# B&R Automation Studio project TD52 (part 17)

```c
/* Source: slatzm.f */
#define slatzm FORTRAN_WRAPPER(slatzm)
extern void slatzm(
    char   *side,
    ptrdiff_t *m,
    ptrdiff_t *n,
    float  *v,
    ptrdiff_t *incv,
    float  *tau,
    float  *c1,
    float  *c2,
    ptrdiff_t *ldc,
    float  *work
);

/* Source: slauu2.f */
#define slauu2 FORTRAN_WRAPPER(slauu2)
extern void slauu2(
    char   *uplo,
    ptrdiff_t *n,
    float  *a,
    ptrdiff_t *lda,
    ptrdiff_t *info
);

/* Source: slauum.f */
#define slauum FORTRAN_WRAPPER(slauum)
extern void slauum(
    char   *uplo,
    ptrdiff_t *n,
    float  *a,
    ptrdiff_t *lda,
    ptrdiff_t *info
);

/* Source: sopgtr.f */
#define sopgtr FORTRAN_WRAPPER(sopgtr)
extern void sopgtr(
    char   *uplo,
    ptrdiff_t *n,
    float  *ap,
    float  *tau,
    float  *q,
    ptrdiff_t *ldq,
    float  *work,
    ptrdiff_t *info
);

/* Source: sopmtr.f */
#define sopmtr FORTRAN_WRAPPER(sopmtr)
extern void sopmtr(
    char   *side,
    char   *uplo,
    char   *trans,
    ptrdiff_t *m,
    ptrdiff_t *n,
    float  *ap,
    float  *tau,
    float  *c,
    ptrdiff_t *ldc,
    float  *work,
    ptrdiff_t *info
);

/* Source: sorg2l.f */
#define sorg2l FORTRAN_WRAPPER(sorg2l)
extern void sorg2l(
    ptrdiff_t *m,
    ptrdiff_t *n,
    ptrdiff_t *k,
    float  *a,
    ptrdiff_t *lda,
    float  *tau,
    float  *work,
    ptrdiff_t *info
);

/* Source: sorg2r.f */
#define sorg2r FORTRAN_WRAPPER(sorg2r)
extern void sorg2r(
    ptrdiff_t *m,
    ptrdiff_t *n,
    ptrdiff_t *k,
    float  *a,
    ptrdiff_t *lda,
    float  *tau,
    float  *work,
    ptrdiff_t *info
);

/* Source: sorgbr.f */
#define sorgbr FORTRAN_WRAPPER(sorgbr)
extern void sorgbr(
    char   *vect,
    ptrdiff_t *m,
    ptrdiff_t *n,
    ptrdiff_t *k,
    float  *a,
    ptrdiff_t *lda,
    float  *tau,
    float  *work,
    ptrdiff_t *lwork,
    ptrdiff_t *info
);

/* Source: sorghr.f */
#define sorghr FORTRAN_WRAPPER(sorghr)
extern void sorghr(
    ptrdiff_t *n,
    ptrdiff_t *ilo,
    ptrdiff_t *ihi,
    float  *a,
    ptrdiff_t *lda,
    float  *tau,
    float  *work,
    ptrdiff_t *lwork,
    ptrdiff_t *info
);

/* Source: sorgl2.f */
#define sorgl2 FORTRAN_WRAPPER(sorgl2)
extern void sorgl2(
    ptrdiff_t *m,
    ptrdiff_t *n,
    ptrdiff_t *k,
    float  *a,
    ptrdiff_t *lda,
    float  *tau,
    float  *work,
    ptrdiff_t *info
);

/* Source: sorglq.f */
#define sorglq FORTRAN_WRAPPER(sorglq)
extern void sorglq(
    ptrdiff_t *m,
    ptrdiff_t *n,
    ptrdiff_t *k,
    float  *a,
    ptrdiff_t *lda,
    float  *tau,
    float  *work,
    ptrdiff_t *lwork,
    ptrdiff_t *info
);

/* Source: sorgql.f */
#define sorgql FORTRAN_WRAPPER(sorgql)
extern void sorgql(
    ptrdiff_t *m,
    ptrdiff_t *n,
    ptrdiff_t *k,
    float  *a,
    ptrdiff_t *lda,
    float  *tau,
    float  *work,
    ptrdiff_t *lwork,
    ptrdiff_t *info
);

/* Source: sorgqr.f */
#define sorgqr FORTRAN_WRAPPER(sorgqr)
extern void sorgqr(
    ptrdiff_t *m,
    ptrdiff_t *n,
    ptrdiff_t *k,
    float  *a,
    ptrdiff_t *lda,
    float  *tau,
    float  *work,
    ptrdiff_t *lwork,
    ptrdiff_t *info
);

/* Source: sorgr2.f */
#define sorgr2 FORTRAN_WRAPPER(sorgr2)
extern void sorgr2(
    ptrdiff_t *m,
    ptrdiff_t *n,
    ptrdiff_t *k,
    float  *a,
    ptrdiff_t *lda,
    float  *tau,
    float  *work,
    ptrdiff_t *info
);

/* Source: sorgrq.f */
#define sorgrq FORTRAN_WRAPPER(sorgrq)
extern void sorgrq(
    ptrdiff_t *m,
    ptrdiff_t *n,
    ptrdiff_t *k,
    float  *a,
    ptrdiff_t *lda,
    float  *tau,
    float  *work,
    ptrdiff_t *lwork,
    ptrdiff_t *info
);

/* Source: sorgtr.f */
#define sorgtr FORTRAN_WRAPPER(sorgtr)
extern void sorgtr(
    char   *uplo,
    ptrdiff_t *n,
    float  *a,
    ptrdiff_t *lda,
    float  *tau,
    float  *work,
    ptrdiff_t *lwork,
    ptrdiff_t *info
);

/* Source: sorm2l.f */
#define sorm2l FORTRAN_WRAPPER(sorm2l)
extern void sorm2l(
    char   *side,
    char   *trans,
    ptrdiff_t *m,
    ptrdiff_t *n,
    ptrdiff_t *k,
    float  *a,
    ptrdiff_t *lda,
    float  *tau,
    float  *c,
    ptrdiff_t *ldc,
    float  *work,
    ptrdiff_t *info
);

/* Source: sorm2r.f */
#define sorm2r FORTRAN_WRAPPER(sorm2r)
extern void sorm2r(
    char   *side,
    char   *trans,
    ptrdiff_t *m,
    ptrdiff_t *n,
    ptrdiff_t *k,
    float  *a,
    ptrdiff_t *lda,
    float  *tau,
    float  *c,
    ptrdiff_t *ldc,
    float  *work,
    ptrdiff_t *info
);

/* Source: sormbr.f */
#define sormbr FORTRAN_WRAPPER(sormbr)
extern void sormbr(
    char   *vect,
    char   *side,
    char   *trans,
    ptrdiff_t *m,
    ptrdiff_t *n,
    ptrdiff_t *k,
    float  *a,
    ptrdiff_t *lda,
    float  *tau,
    float  *c,
    ptrdiff_t *ldc,
    float  *work,
    ptrdiff_t *lwork,
    ptrdiff_t *info
);

/* Source: sormhr.f */
#define sormhr FORTRAN_WRAPPER(sormhr)
extern void sormhr(
    char   *side,
    char   *trans,
    ptrdiff_t *m,
    ptrdiff_t *n,
    ptrdiff_t *ilo,
    ptrdiff_t *ihi,
    float  *a,
    ptrdiff_t *lda,
    float  *tau,
    float  *c,
    ptrdiff_t *ldc,
    float  *work,
    ptrdiff_t *lwork,
    ptrdiff_t *info
);

/* Source: sorml2.f */
#define sorml2 FORTRAN_WRAPPER(sorml2)
extern void sorml2(
    char   *side,
    char   *trans,
    ptrdiff_t *m,
    ptrdiff_t *n,
    ptrdiff_t *k,
    float  *a,
    ptrdiff_t *lda,
    float  *tau,
    float  *c,
    ptrdiff_t *ldc,
    float  *work,
    ptrdiff_t *info
);

/* Source: sormlq.f */
#define sormlq FORTRAN_WRAPPER(sormlq)
extern void sormlq(
    char   *side,
    char   *trans,
    ptrdiff_t *m,
    ptrdiff_t *n,
    ptrdiff_t *k,
    float  *a,
    ptrdiff_t *lda,
    float  *tau,
    float  *c,
    ptrdiff_t *ldc,
    float  *work,
    ptrdiff_t *lwork,
    ptrdiff_t *info
);

/* Source: sormql.f */
#define sormql FORTRAN_WRAPPER(sormql)
extern void sormql(
    char   *side,
    char   *trans,
    ptrdiff_t *m,
    ptrdiff_t *n,
    ptrdiff_t *k,
    float  *a,
    ptrdiff_t *lda,
    float  *tau,
    float  *c,
    ptrdiff_t *ldc,
    float  *work,
    ptrdiff_t *lwork,
    ptrdiff_t *info
);

/* Source: sormqr.f */
#define sormqr FORTRAN_WRAPPER(sormqr)
extern void sormqr(
    char   *side,
    char   *trans,
    ptrdiff_t *m,
    ptrdiff_t *n,
    ptrdiff_t *k,
    float  *a,
    ptrdiff_t *lda,
    float  *tau,
    float  *c,
    ptrdiff_t *ldc,
    float  *work,
    ptrdiff_t *lwork,
    ptrdiff_t *info
);

/* Source: sormr2.f */
#define sormr2 FORTRAN_WRAPPER(sormr2)
extern void sormr2(
    char   *side,
    char   *trans,
    ptrdiff_t *m,
    ptrdiff_t *n,
    ptrdiff_t *k,
    float  *a,
    ptrdiff_t *lda,
    float  *tau,
    float  *c,
    ptrdiff_t *ldc,
    float  *work,
    ptrdiff_t *info
);

/* Source: sormr3.f */
#define sormr3 FORTRAN_WRAPPER(sormr3)
extern void sormr3(
    char   *side,
    char   *trans,
    ptrdiff_t *m,
    ptrdiff_t *n,
    ptrdiff_t *k,
    ptrdiff_t *l,
    float  *a,
    ptrdiff_t *lda,
    float  *tau,
    float  *c,
    ptrdiff_t *ldc,
    float  *work,
    ptrdiff_t *info
);

/* Source: sormrq.f */
#define sormrq FORTRAN_WRAPPER(sormrq)
extern void sormrq(
    char   *side,
    char   *trans,
    ptrdiff_t *m,
    ptrdiff_t *n,
    ptrdiff_t *k,
    float  *a,
    ptrdiff_t *lda,
    float  *tau,
    float  *c,
    ptrdiff_t *ldc,
    float  *work,
    ptrdiff_t *lwork,
    ptrdiff_t *info
);

/* Source: sormrz.f */
#define sormrz FORTRAN_WRAPPER(sormrz)
extern void sormrz(
    char   *side,
    char   *trans,
    ptrdiff_t *m,
    ptrdiff_t *n,
    ptrdiff_t *k,
    ptrdiff_t *l,
    float  *a,
    ptrdiff_t *lda,
    float  *tau,
    float  *c,
    ptrdiff_t *ldc,
    float  *work,
    ptrdiff_t *lwork,
    ptrdiff_t *info
);

/* Source: sormtr.f */
#define sormtr FORTRAN_WRAPPER(sormtr)
extern void sormtr(
    char   *side,
    char   *uplo,
    char   *trans,
    ptrdiff_t *m,
    ptrdiff_t *n,
    float  *a,
    ptrdiff_t *lda,
    float  *tau,
    float  *c,
    ptrdiff_t *ldc,
    float  *work,
    ptrdiff_t *lwork,
    ptrdiff_t *info
);

/* Source: spbcon.f */
#define spbcon FORTRAN_WRAPPER(spbcon)
extern void spbcon(
    char   *uplo,
    ptrdiff_t *n,
    ptrdiff_t *kd,
    float  *ab,
    ptrdiff_t *ldab,
    float  *anorm,
    float  *rcond,
    float  *work,
    ptrdiff_t *iwork,
    ptrdiff_t *info
);

/* Source: spbequ.f */
#define spbequ FORTRAN_WRAPPER(spbequ)
extern void spbequ(
    char   *uplo,
    ptrdiff_t *n,
    ptrdiff_t *kd,
    float  *ab,
    ptrdiff_t *ldab,
    float  *s,
    float  *scond,
    float  *amax,
    ptrdiff_t *info
);

/* Source: spbrfs.f */
#define spbrfs FORTRAN_WRAPPER(spbrfs)
extern void spbrfs(
    char   *uplo,
    ptrdiff_t *n,
    ptrdiff_t *kd,
    ptrdiff_t *nrhs,
    float  *ab,
    ptrdiff_t *ldab,
    float  *afb,
    ptrdiff_t *ldafb,
    float  *b,
    ptrdiff_t *ldb,
    float  *x,
    ptrdiff_t *ldx,
    float  *ferr,
    float  *berr,
    float  *work,
    ptrdiff_t *iwork,
    ptrdiff_t *info
);

/* Source: spbstf.f */
#define spbstf FORTRAN_WRAPPER(spbstf)
extern void spbstf(
    char   *uplo,
    ptrdiff_t *n,
    ptrdiff_t *kd,
    float  *ab,
    ptrdiff_t *ldab,
    ptrdiff_t *info
);

/* Source: spbsv.f */
#define spbsv FORTRAN_WRAPPER(spbsv)
extern void spbsv(
    char   *uplo,
    ptrdiff_t *n,
    ptrdiff_t *kd,
    ptrdiff_t *nrhs,
    float  *ab,
    ptrdiff_t *ldab,
    float  *b,
    ptrdiff_t *ldb,
    ptrdiff_t *info
);

/* Source: spbsvx.f */
#define spbsvx FORTRAN_WRAPPER(spbsvx)
extern void spbsvx(
    char   *fact,
    char   *uplo,
    ptrdiff_t *n,
    ptrdiff_t *kd,
    ptrdiff_t *nrhs,
    float  *ab,
    ptrdiff_t *ldab,
    float  *afb,
    ptrdiff_t *ldafb,
    char   *equed,
    float  *s,
    float  *b,
    ptrdiff_t *ldb,
    float  *x,
    ptrdiff_t *ldx,
    float  *rcond,
    float  *ferr,
    float  *berr,
    float  *work,
    ptrdiff_t *iwork,
    ptrdiff_t *info
);

/* Source: spbtf2.f */
#define spbtf2 FORTRAN_WRAPPER(spbtf2)
extern void spbtf2(
    char   *uplo,
    ptrdiff_t *n,
    ptrdiff_t *kd,
    float  *ab,
    ptrdiff_t *ldab,
    ptrdiff_t *info
);

/* Source: spbtrf.f */
#define spbtrf FORTRAN_WRAPPER(spbtrf)
extern void spbtrf(
    char   *uplo,
    ptrdiff_t *n,
    ptrdiff_t *kd,
    float  *ab,
    ptrdiff_t *ldab,
    ptrdiff_t *info
);

/* Source: spbtrs.f */
#define spbtrs FORTRAN_WRAPPER(spbtrs)
extern void spbtrs(
    char   *uplo,
    ptrdiff_t *n,
    ptrdiff_t *kd,
    ptrdiff_t *nrhs,
    float  *ab,
    ptrdiff_t *ldab,
    float  *b,
    ptrdiff_t *ldb,
    ptrdiff_t *info
);

/* Source: spftrf.f */
#define spftrf FORTRAN_WRAPPER(spftrf)
extern void spftrf(
    char   *transr,
    char   *uplo,
    ptrdiff_t *n,
    float  *a,
    ptrdiff_t *info
);

/* Source: spftri.f */
#define spftri FORTRAN_WRAPPER(spftri)
extern void spftri(
    char   *transr,
    char   *uplo,
    ptrdiff_t *n,
    float  *a,
    ptrdiff_t *info
);

/* Source: spftrs.f */
#define spftrs FORTRAN_WRAPPER(spftrs)
extern void spftrs(
    char   *transr,
    char   *uplo,
    ptrdiff_t *n,
    ptrdiff_t *nrhs,
    float  *a,
    float  *b,
    ptrdiff_t *ldb,
    ptrdiff_t *info
);

/* Source: spocon.f */
#define spocon FORTRAN_WRAPPER(spocon)
extern void spocon(
    char   *uplo,
    ptrdiff_t *n,
    float  *a,
    ptrdiff_t *lda,
    float  *anorm,
    float  *rcond,
    float  *work,
    ptrdiff_t *iwork,
    ptrdiff_t *info
);

/* Source: spoequ.f */
#define spoequ FORTRAN_WRAPPER(spoequ)
extern void spoequ(
    ptrdiff_t *n,
    float  *a,
    ptrdiff_t *lda,
    float  *s,
    float  *scond,
    float  *amax,
    ptrdiff_t *info
);

/* Source: spoequb.f */
#define spoequb FORTRAN_WRAPPER(spoequb)
extern void spoequb(
    ptrdiff_t *n,
    float  *a,
    ptrdiff_t *lda,
    float  *s,
    float  *scond,
    float  *amax,
    ptrdiff_t *info
);

/* Source: sporfs.f */
#define sporfs FORTRAN_WRAPPER(sporfs)
extern void sporfs(
    char   *uplo,
    ptrdiff_t *n,
    ptrdiff_t *nrhs,
    float  *a,
    ptrdiff_t *lda,
    float  *af,
    ptrdiff_t *ldaf,
    float  *b,
    ptrdiff_t *ldb,
    float  *x,
    ptrdiff_t *ldx,
    float  *ferr,
    float  *berr,
    float  *work,
    ptrdiff_t *iwork,
    ptrdiff_t *info
);

/* Source: sposv.f */
#define sposv FORTRAN_WRAPPER(sposv)
extern void sposv(
    char   *uplo,
    ptrdiff_t *n,
    ptrdiff_t *nrhs,
    float  *a,
    ptrdiff_t *lda,
    float  *b,
    ptrdiff_t *ldb,
    ptrdiff_t *info
);

/* Source: sposvx.f */
#define sposvx FORTRAN_WRAPPER(sposvx)
extern void sposvx(
    char   *fact,
    char   *uplo,
    ptrdiff_t *n,
    ptrdiff_t *nrhs,
    float  *a,
    ptrdiff_t *lda,
    float  *af,
    ptrdiff_t *ldaf,
    char   *equed,
    float  *s,
    float  *b,
    ptrdiff_t *ldb,
    float  *x,
    ptrdiff_t *ldx,
    float  *rcond,
    float  *ferr,
    float  *berr,
    float  *work,
    ptrdiff_t *iwork,
    ptrdiff_t *info
);

/* Source: spotf2.f */
#define spotf2 FORTRAN_WRAPPER(spotf2)
extern void spotf2(
    char   *uplo,
    ptrdiff_t *n,
    float  *a,
    ptrdiff_t *lda,
    ptrdiff_t *info
);

/* Source: spotrf.f */
#define spotrf FORTRAN_WRAPPER(spotrf)
extern void spotrf(
    char   *uplo,
    ptrdiff_t *n,
    float  *a,
    ptrdiff_t *lda,
    ptrdiff_t *info
);

/* Source: spotri.f */
#define spotri FORTRAN_WRAPPER(spotri)
extern void spotri(
    char   *uplo,
    ptrdiff_t *n,
    float  *a,
    ptrdiff_t *lda,
    ptrdiff_t *info
);

/* Source: spotrs.f */
#define spotrs FORTRAN_WRAPPER(spotrs)
extern void spotrs(
    char   *uplo,
    ptrdiff_t *n,
    ptrdiff_t *nrhs,
    float  *a,
    ptrdiff_t *lda,
    float  *b,
    ptrdiff_t *ldb,
    ptrdiff_t *info
);

/* Source: sppcon.f */
#define sppcon FORTRAN_WRAPPER(sppcon)
extern void sppcon(
    char   *uplo,
    ptrdiff_t *n,
    float  *ap,
    float  *anorm,
    float  *rcond,
    float  *work,
    ptrdiff_t *iwork,
    ptrdiff_t *info
);

/* Source: sppequ.f */
#define sppequ FORTRAN_WRAPPER(sppequ)
extern void sppequ(
    char   *uplo,
    ptrdiff_t *n,
    float  *ap,
    float  *s,
    float  *scond,
    float  *amax,
    ptrdiff_t *info
);

/* Source: spprfs.f */
#define spprfs FORTRAN_WRAPPER(spprfs)
extern void spprfs(
    char   *uplo,
    ptrdiff_t *n,
    ptrdiff_t *nrhs,
    float  *ap,
    float  *afp,
    float  *b,
    ptrdiff_t *ldb,
    float  *x,
    ptrdiff_t *ldx,
    float  *ferr,
    float  *berr,
    float  *work,
    ptrdiff_t *iwork,
    ptrdiff_t *info
);

/* Source: sppsv.f */
#define sppsv FORTRAN_WRAPPER(sppsv)
extern void sppsv(
    char   *uplo,
    ptrdiff_t *n,
    ptrdiff_t *nrhs,
    float  *ap,
    float  *b,
    ptrdiff_t *ldb,
    ptrdiff_t *info
);

/* Source: sppsvx.f */
#define sppsvx FORTRAN_WRAPPER(sppsvx)
extern void sppsvx(
    char   *fact,
    char   *uplo,
    ptrdiff_t *n,
    ptrdiff_t *nrhs,
    float  *ap,
    float  *afp,
    char   *equed,
    float  *s,
    float  *b,
    ptrdiff_t *ldb,
    float  *x,
    ptrdiff_t *ldx,
    float  *rcond,
    float  *ferr,
    float  *berr,
    float  *work,
    ptrdiff_t *iwork,
    ptrdiff_t *info
);

/* Source: spptrf.f */
#define spptrf FORTRAN_WRAPPER(spptrf)
extern void spptrf(
    char   *uplo,
    ptrdiff_t *n,
    float  *ap,
    ptrdiff_t *info
);

/* Source: spptri.f */
#define spptri FORTRAN_WRAPPER(spptri)
extern void spptri(
    char   *uplo,
    ptrdiff_t *n,
    float  *ap,
    ptrdiff_t *info
);

/* Source: spptrs.f */
#define spptrs FORTRAN_WRAPPER(spptrs)
extern void spptrs(
    char   *uplo,
    ptrdiff_t *n,
    ptrdiff_t *nrhs,
    float  *ap,
    float  *b,
    ptrdiff_t *ldb,
    ptrdiff_t *info
);

/* Source: spstf2.f */
#define spstf2 FORTRAN_WRAPPER(spstf2)
extern void spstf2(
    char   *uplo,
    ptrdiff_t *n,
    float  *a,
    ptrdiff_t *lda,
    ptrdiff_t *piv,
    ptrdiff_t *rank,
    float  *tol,
    float  *work,
    ptrdiff_t *info
);

/* Source: spstrf.f */
#define spstrf FORTRAN_WRAPPER(spstrf)
extern void spstrf(
    char   *uplo,
    ptrdiff_t *n,
    float  *a,
    ptrdiff_t *lda,
    ptrdiff_t *piv,
    ptrdiff_t *rank,
    float  *tol,
    float  *work,
    ptrdiff_t *info
);

/* Source: sptcon.f */
#define sptcon FORTRAN_WRAPPER(sptcon)
extern void sptcon(
    ptrdiff_t *n,
    float  *d,
    float  *e,
    float  *anorm,
    float  *rcond,
    float  *work,
    ptrdiff_t *info
);

/* Source: spteqr.f */
#define spteqr FORTRAN_WRAPPER(spteqr)
extern void spteqr(
    char   *compz,
    ptrdiff_t *n,
    float  *d,
    float  *e,
    float  *z,
    ptrdiff_t *ldz,
    float  *work,
    ptrdiff_t *info
);

/* Source: sptrfs.f */
#define sptrfs FORTRAN_WRAPPER(sptrfs)
extern void sptrfs(
    ptrdiff_t *n,
    ptrdiff_t *nrhs,
    float  *d,
    float  *e,
    float  *df,
    float  *ef,
    float  *b,
    ptrdiff_t *ldb,
    float  *x,
    ptrdiff_t *ldx,
    float  *ferr,
    float  *berr,
    float  *work,
    ptrdiff_t *info
);

/* Source: sptsv.f */
#define sptsv FORTRAN_WRAPPER(sptsv)
extern void sptsv(
    ptrdiff_t *n,
    ptrdiff_t *nrhs,
    float  *d,
    float  *e,
    float  *b,
    ptrdiff_t *ldb,
    ptrdiff_t *info
);

/* Source: sptsvx.f */
#define sptsvx FORTRAN_WRAPPER(sptsvx)
extern void sptsvx(
    char   *fact,
    ptrdiff_t *n,
    ptrdiff_t *nrhs,
    float  *d,
    float  *e,
    float  *df,
    float  *ef,
    float  *b,
    ptrdiff_t *ldb,
    float  *x,
    ptrdiff_t *ldx,
    float  *rcond,
    float  *ferr,
    float  *berr,
    float  *work,
    ptrdiff_t *info
);

/* Source: spttrf.f */
#define spttrf FORTRAN_WRAPPER(spttrf)
extern void spttrf(
    ptrdiff_t *n,
    float  *d,
    float  *e,
    ptrdiff_t *info
);

/* Source: spttrs.f */
#define spttrs FORTRAN_WRAPPER(spttrs)
extern void spttrs(
    ptrdiff_t *n,
    ptrdiff_t *nrhs,
    float  *d,
    float  *e,
    float  *b,
    ptrdiff_t *ldb,
    ptrdiff_t *info
);

/* Source: sptts2.f */
#define sptts2 FORTRAN_WRAPPER(sptts2)
extern void sptts2(
    ptrdiff_t *n,
    ptrdiff_t *nrhs,
    float  *d,
    float  *e,
    float  *b,
    ptrdiff_t *ldb
);

/* Source: srscl.f */
#define srscl FORTRAN_WRAPPER(srscl)
extern void srscl(
    ptrdiff_t *n,
    float  *sa,
    float  *sx,
    ptrdiff_t *incx
);

/* Source: ssbev.f */
#define ssbev FORTRAN_WRAPPER(ssbev)
extern void ssbev(
    char   *jobz,
    char   *uplo,
    ptrdiff_t *n,
    ptrdiff_t *kd,
    float  *ab,
    ptrdiff_t *ldab,
    float  *w,
    float  *z,
    ptrdiff_t *ldz,
    float  *work,
    ptrdiff_t *info
);

/* Source: ssbevd.f */
#define ssbevd FORTRAN_WRAPPER(ssbevd)
extern void ssbevd(
    char   *jobz,
    char   *uplo,
    ptrdiff_t *n,
    ptrdiff_t *kd,
    float  *ab,
    ptrdiff_t *ldab,
    float  *w,
    float  *z,
    ptrdiff_t *ldz,
    float  *work,
    ptrdiff_t *lwork,
    ptrdiff_t *iwork,
    ptrdiff_t *liwork,
    ptrdiff_t *info
);

/* Source: ssbevx.f */
#define ssbevx FORTRAN_WRAPPER(ssbevx)
extern void ssbevx(
    char   *jobz,
    char   *range,
    char   *uplo,
    ptrdiff_t *n,
    ptrdiff_t *kd,
    float  *ab,
    ptrdiff_t *ldab,
    float  *q,
    ptrdiff_t *ldq,
    float  *vl,
    float  *vu,
    ptrdiff_t *il,
    ptrdiff_t *iu,
    float  *abstol,
    ptrdiff_t *m,
    float  *w,
    float  *z,
    ptrdiff_t *ldz,
    float  *work,
    ptrdiff_t *iwork,
    ptrdiff_t *ifail,
    ptrdiff_t *info
);

/* Source: ssbgst.f */
#define ssbgst FORTRAN_WRAPPER(ssbgst)
extern void ssbgst(
    char   *vect,
    char   *uplo,
    ptrdiff_t *n,
    ptrdiff_t *ka,
    ptrdiff_t *kb,
    float  *ab,
    ptrdiff_t *ldab,
    float  *bb,
    ptrdiff_t *ldbb,
    float  *x,
    ptrdiff_t *ldx,
    float  *work,
    ptrdiff_t *info
);

/* Source: ssbgv.f */
#define ssbgv FORTRAN_WRAPPER(ssbgv)
extern void ssbgv(
    char   *jobz,
    char   *uplo,
    ptrdiff_t *n,
    ptrdiff_t *ka,
    ptrdiff_t *kb,
    float  *ab,
    ptrdiff_t *ldab,
    float  *bb,
    ptrdiff_t *ldbb,
    float  *w,
    float  *z,
    ptrdiff_t *ldz,
    float  *work,
    ptrdiff_t *info
);

/* Source: ssbgvd.f */
#define ssbgvd FORTRAN_WRAPPER(ssbgvd)
extern void ssbgvd(
    char   *jobz,
    char   *uplo,
    ptrdiff_t *n,
    ptrdiff_t *ka,
    ptrdiff_t *kb,
    float  *ab,
    ptrdiff_t *ldab,
    float  *bb,
    ptrdiff_t *ldbb,
    float  *w,
    float  *z,
    ptrdiff_t *ldz,
    float  *work,
    ptrdiff_t *lwork,
    ptrdiff_t *iwork,
    ptrdiff_t *liwork,
    ptrdiff_t *info
);

/* Source: ssbgvx.f */
#define ssbgvx FORTRAN_WRAPPER(ssbgvx)
extern void ssbgvx(
    char   *jobz,
    char   *range,
    char   *uplo,
    ptrdiff_t *n,
    ptrdiff_t *ka,
    ptrdiff_t *kb,
    float  *ab,
    ptrdiff_t *ldab,
    float  *bb,
    ptrdiff_t *ldbb,
    float  *q,
    ptrdiff_t *ldq,
    float  *vl,
    float  *vu,
    ptrdiff_t *il,
    ptrdiff_t *iu,
    float  *abstol,
    ptrdiff_t *m,
    float  *w,
    float  *z,
    ptrdiff_t *ldz,
    float  *work,
    ptrdiff_t *iwork,
    ptrdiff_t *ifail,
    ptrdiff_t *info
);

/* Source: ssbtrd.f */
#define ssbtrd FORTRAN_WRAPPER(ssbtrd)
extern void ssbtrd(
    char   *vect,
    char   *uplo,
    ptrdiff_t *n,
    ptrdiff_t *kd,
    float  *ab,
    ptrdiff_t *ldab,
    float  *d,
    float  *e,
    float  *q,
    ptrdiff_t *ldq,
    float  *work,
    ptrdiff_t *info
);

/* Source: ssfrk.f */
#define ssfrk FORTRAN_WRAPPER(ssfrk)
extern void ssfrk(
    char   *transr,
    char   *uplo,
    char   *trans,
    ptrdiff_t *n,
    ptrdiff_t *k,
    float  *alpha,
    float  *a,
    ptrdiff_t *lda,
    float  *beta,
    float  *c
);

/* Source: sspcon.f */
#define sspcon FORTRAN_WRAPPER(sspcon)
extern void sspcon(
    char   *uplo,
    ptrdiff_t *n,
    float  *ap,
    ptrdiff_t *ipiv,
    float  *anorm,
    float  *rcond,
    float  *work,
    ptrdiff_t *iwork,
    ptrdiff_t *info
);

/* Source: sspev.f */
#define sspev FORTRAN_WRAPPER(sspev)
extern void sspev(
    char   *jobz,
    char   *uplo,
    ptrdiff_t *n,
    float  *ap,
    float  *w,
    float  *z,
    ptrdiff_t *ldz,
    float  *work,
    ptrdiff_t *info
);

/* Source: sspevd.f */
#define sspevd FORTRAN_WRAPPER(sspevd)
extern void sspevd(
    char   *jobz,
    char   *uplo,
    ptrdiff_t *n,
    float  *ap,
    float  *w,
    float  *z,
    ptrdiff_t *ldz,
    float  *work,
    ptrdiff_t *lwork,
    ptrdiff_t *iwork,
    ptrdiff_t *liwork,
    ptrdiff_t *info
);

/* Source: sspevx.f */
#define sspevx FORTRAN_WRAPPER(sspevx)
extern void sspevx(
    char   *jobz,
    char   *range,
    char   *uplo,
    ptrdiff_t *n,
    float  *ap,
    float  *vl,
    float  *vu,
    ptrdiff_t *il,
    ptrdiff_t *iu,
    float  *abstol,
    ptrdiff_t *m,
    float  *w,
    float  *z,
    ptrdiff_t *ldz,
    float  *work,
    ptrdiff_t *iwork,
    ptrdiff_t *ifail,
    ptrdiff_t *info
);

/* Source: sspgst.f */
#define sspgst FORTRAN_WRAPPER(sspgst)
extern void sspgst(
    ptrdiff_t *itype,
    char   *uplo,
    ptrdiff_t *n,
    float  *ap,
    float  *bp,
    ptrdiff_t *info
);

/* Source: sspgv.f */
#define sspgv FORTRAN_WRAPPER(sspgv)
extern void sspgv(
    ptrdiff_t *itype,
    char   *jobz,
    char   *uplo,
    ptrdiff_t *n,
    float  *ap,
    float  *bp,
    float  *w,
    float  *z,
    ptrdiff_t *ldz,
    float  *work,
    ptrdiff_t *info
);

/* Source: sspgvd.f */
#define sspgvd FORTRAN_WRAPPER(sspgvd)
extern void sspgvd(
    ptrdiff_t *itype,
    char   *jobz,
    char   *uplo,
    ptrdiff_t *n,
    float  *ap,
    float  *bp,
    float  *w,
    float  *z,
    ptrdiff_t *ldz,
    float  *work,
    ptrdiff_t *lwork,
    ptrdiff_t *iwork,
    ptrdiff_t *liwork,
    ptrdiff_t *info
);

/* Source: sspgvx.f */
#define sspgvx FORTRAN_WRAPPER(sspgvx)
extern void sspgvx(
    ptrdiff_t *itype,
    char   *jobz,
    char   *range,
    char   *uplo,
    ptrdiff_t *n,
    float  *ap,
    float  *bp,
    float  *vl,
    float  *vu,
    ptrdiff_t *il,
    ptrdiff_t *iu,
    float  *abstol,
    ptrdiff_t *m,
    float  *w,
    float  *z,
    ptrdiff_t *ldz,
    float  *work,
    ptrdiff_t *iwork,
    ptrdiff_t *ifail,
    ptrdiff_t *info
);

/* Source: ssprfs.f */
#define ssprfs FORTRAN_WRAPPER(ssprfs)
extern void ssprfs(
    char   *uplo,
    ptrdiff_t *n,
    ptrdiff_t *nrhs,
    float  *ap,
    float  *afp,
    ptrdiff_t *ipiv,
    float  *b,
    ptrdiff_t *ldb,
    float  *x,
    ptrdiff_t *ldx,
    float  *ferr,
    float  *berr,
    float  *work,
    ptrdiff_t *iwork,
    ptrdiff_t *info
);

/* Source: sspsv.f */
#define sspsv FORTRAN_WRAPPER(sspsv)
extern void sspsv(
    char   *uplo,
    ptrdiff_t *n,
    ptrdiff_t *nrhs,
    float  *ap,
    ptrdiff_t *ipiv,
    float  *b,
    ptrdiff_t *ldb,
    ptrdiff_t *info
);

/* Source: sspsvx.f */
#define sspsvx FORTRAN_WRAPPER(sspsvx)
extern void sspsvx(
    char   *fact,
    char   *uplo,
    ptrdiff_t *n,
    ptrdiff_t *nrhs,
    float  *ap,
    float  *afp,
    ptrdiff_t *ipiv,
    float  *b,
    ptrdiff_t *ldb,
    float  *x,
    ptrdiff_t *ldx,
    float  *rcond,
    float  *ferr,
    float  *berr,
    float  *work,
    ptrdiff_t *iwork,
    ptrdiff_t *info
);

/* Source: ssptrd.f */
#define ssptrd FORTRAN_WRAPPER(ssptrd)
extern void ssptrd(
    char   *uplo,
    ptrdiff_t *n,
    float  *ap,
    float  *d,
    float  *e,
    float  *tau,
    ptrdiff_t *info
);

/* Source: ssptrf.f */
#define ssptrf FORTRAN_WRAPPER(ssptrf)
extern void ssptrf(
    char   *uplo,
    ptrdiff_t *n,
    float  *ap,
    ptrdiff_t *ipiv,
    ptrdiff_t *info
);

/* Source: ssptri.f */
#define ssptri FORTRAN_WRAPPER(ssptri)
extern void ssptri(
    char   *uplo,
    ptrdiff_t *n,
    float  *ap,
    ptrdiff_t *ipiv,
    float  *work,
    ptrdiff_t *info
);

/* Source: ssptrs.f */
#define ssptrs FORTRAN_WRAPPER(ssptrs)
extern void ssptrs(
    char   *uplo,
    ptrdiff_t *n,
    ptrdiff_t *nrhs,
    float  *ap,
    ptrdiff_t *ipiv,
    float  *b,
    ptrdiff_t *ldb,
    ptrdiff_t *info
);

/* Source: sstebz.f */
#define sstebz FORTRAN_WRAPPER(sstebz)
extern void sstebz(
    char   *range,
    char   *order,
    ptrdiff_t *n,
    float  *vl,
    float  *vu,
    ptrdiff_t *il,
    ptrdiff_t *iu,
    float  *abstol,
    float  *d,
    float  *e,
    ptrdiff_t *m,
    ptrdiff_t *nsplit,
    float  *w,
    ptrdiff_t *iblock,
    ptrdiff_t *isplit,
    float  *work,
    ptrdiff_t *iwork,
    ptrdiff_t *info
);

/* Source: sstedc.f */
#define sstedc FORTRAN_WRAPPER(sstedc)
extern void sstedc(
    char   *compz,
    ptrdiff_t *n,
    float  *d,
    float  *e,
    float  *z,
    ptrdiff_t *ldz,
    float  *work,
    ptrdiff_t *lwork,
    ptrdiff_t *iwork,
    ptrdiff_t *liwork,
    ptrdiff_t *info
);

/* Source: sstegr.f */
#define sstegr FORTRAN_WRAPPER(sstegr)
extern void sstegr(
    char   *jobz,
    char   *range,
    ptrdiff_t *n,
    float  *d,
    float  *e,
    float  *vl,
    float  *vu,
    ptrdiff_t *il,
    ptrdiff_t *iu,
    float  *abstol,
    ptrdiff_t *m,
    float  *w,
    float  *z,
    ptrdiff_t *ldz,
    ptrdiff_t *isuppz,
    float  *work,
    ptrdiff_t *lwork,
    ptrdiff_t *iwork,
    ptrdiff_t *liwork,
    ptrdiff_t *info
);

/* Source: sstein.f */
#define sstein FORTRAN_WRAPPER(sstein)
extern void sstein(
    ptrdiff_t *n,
    float  *d,
    float  *e,
    ptrdiff_t *m,
    float  *w,
    ptrdiff_t *iblock,
    ptrdiff_t *isplit,
    float  *z,
    ptrdiff_t *ldz,
    float  *work,
    ptrdiff_t *iwork,
    ptrdiff_t *ifail,
    ptrdiff_t *info
);

/* Source: sstemr.f */
#define sstemr FORTRAN_WRAPPER(sstemr)
extern void sstemr(
    char   *jobz,
    char   *range,
    ptrdiff_t *n,
    float  *d,
    float  *e,
    float  *vl,
    float  *vu,
    ptrdiff_t *il,
    ptrdiff_t *iu,
    ptrdiff_t *m,
    float  *w,
    float  *z,
    ptrdiff_t *ldz,
    ptrdiff_t *nzc,
    ptrdiff_t *isuppz,
    ptrdiff_t *tryrac,
    float  *work,
    ptrdiff_t *lwork,
    ptrdiff_t *iwork,
    ptrdiff_t *liwork,
    ptrdiff_t *info
);

/* Source: ssteqr.f */
#define ssteqr FORTRAN_WRAPPER(ssteqr)
extern void ssteqr(
    char   *compz,
    ptrdiff_t *n,
    float  *d,
    float  *e,
    float  *z,
    ptrdiff_t *ldz,
    float  *work,
    ptrdiff_t *info
);

/* Source: ssterf.f */
#define ssterf FORTRAN_WRAPPER(ssterf)
extern void ssterf(
    ptrdiff_t *n,
    float  *d,
    float  *e,
    ptrdiff_t *info
);

/* Source: sstev.f */
#define sstev FORTRAN_WRAPPER(sstev)
extern void sstev(
    char   *jobz,
    ptrdiff_t *n,
    float  *d,
    float  *e,
    float  *z,
    ptrdiff_t *ldz,
    float  *work,
    ptrdiff_t *info
);

/* Source: sstevd.f */
#define sstevd FORTRAN_WRAPPER(sstevd)
extern void sstevd(
    char   *jobz,
    ptrdiff_t *n,
    float  *d,
    float  *e,
    float  *z,
    ptrdiff_t *ldz,
    float  *work,
    ptrdiff_t *lwork,
    ptrdiff_t *iwork,
    ptrdiff_t *liwork,
    ptrdiff_t *info
);

/* Source: sstevr.f */
#define sstevr FORTRAN_WRAPPER(sstevr)
extern void sstevr(
    char   *jobz,
    char   *range,
    ptrdiff_t *n,
    float  *d,
    float  *e,
    float  *vl,
    float  *vu,
    ptrdiff_t *il,
    ptrdiff_t *iu,
    float  *abstol,
    ptrdiff_t *m,
    float  *w,
    float  *z,
    ptrdiff_t *ldz,
    ptrdiff_t *isuppz,
    float  *work,
    ptrdiff_t *lwork,
    ptrdiff_t *iwork,
    ptrdiff_t *liwork,
    ptrdiff_t *info
);

/* Source: sstevx.f */
#define sstevx FORTRAN_WRAPPER(sstevx)
extern void sstevx(
    char   *jobz,
    char   *range,
    ptrdiff_t *n,
    float  *d,
    float  *e,
    float  *vl,
    float  *vu,
    ptrdiff_t *il,
    ptrdiff_t *iu,
    float  *abstol,
    ptrdiff_t *m,
    float  *w,
    float  *z,
    ptrdiff_t *ldz,
    float  *work,
    ptrdiff_t *iwork,
    ptrdiff_t *ifail,
    ptrdiff_t *info
);

/* Source: ssycon.f */
#define ssycon FORTRAN_WRAPPER(ssycon)
extern void ssycon(
    char   *uplo,
    ptrdiff_t *n,
    float  *a,
    ptrdiff_t *lda,
    ptrdiff_t *ipiv,
    float  *anorm,
    float  *rcond,
    float  *work,
    ptrdiff_t *iwork,
    ptrdiff_t *info
);

/* Source: ssyequb.f */
#define ssyequb FORTRAN_WRAPPER(ssyequb)
extern void ssyequb(
    char   *uplo,
    ptrdiff_t *n,
    float  *a,
    ptrdiff_t *lda,
    float  *s,
    float  *scond,
    float  *amax,
    float  *work,
    ptrdiff_t *info
);

/* Source: ssyev.f */
#define ssyev FORTRAN_WRAPPER(ssyev)
extern void ssyev(
    char   *jobz,
    char   *uplo,
    ptrdiff_t *n,
    float  *a,
    ptrdiff_t *lda,
    float  *w,
    float  *work,
    ptrdiff_t *lwork,
    ptrdiff_t *info
);

/* Source: ssyevd.f */
#define ssyevd FORTRAN_WRAPPER(ssyevd)
extern void ssyevd(
    char   *jobz,
    char   *uplo,
    ptrdiff_t *n,
    float  *a,
    ptrdiff_t *lda,
    float  *w,
    float  *work,
    ptrdiff_t *lwork,
    ptrdiff_t *iwork,
    ptrdiff_t *liwork,
    ptrdiff_t *info
);

/* Source: ssyevr.f */
#define ssyevr FORTRAN_WRAPPER(ssyevr)
extern void ssyevr(
    char   *jobz,
    char   *range,
    char   *uplo,
    ptrdiff_t *n,
    float  *a,
    ptrdiff_t *lda,
    float  *vl,
    float  *vu,
    ptrdiff_t *il,
    ptrdiff_t *iu,
    float  *abstol,
    ptrdiff_t *m,
    float  *w,
    float  *z,
    ptrdiff_t *ldz,
    ptrdiff_t *isuppz,
    float  *work,
    ptrdiff_t *lwork,
    ptrdiff_t *iwork,
    ptrdiff_t *liwork,
    ptrdiff_t *info
);

/* Source: ssyevx.f */
#define ssyevx FORTRAN_WRAPPER(ssyevx)
extern void ssyevx(
    char   *jobz,
    char   *range,
    char   *uplo,
    ptrdiff_t *n,
    float  *a,
    ptrdiff_t *lda,
    float  *vl,
    float  *vu,
    ptrdiff_t *il,
    ptrdiff_t *iu,
    float  *abstol,
    ptrdiff_t *m,
    float  *w,
    float  *z,
    ptrdiff_t *ldz,
    float  *work,
    ptrdiff_t *lwork,
    ptrdiff_t *iwork,
    ptrdiff_t *ifail,
    ptrdiff_t *info
);

/* Source: ssygs2.f */
#define ssygs2 FORTRAN_WRAPPER(ssygs2)
extern void ssygs2(
    ptrdiff_t *itype,
    char   *uplo,
    ptrdiff_t *n,
    float  *a,
    ptrdiff_t *lda,
    float  *b,
    ptrdiff_t *ldb,
    ptrdiff_t *info
);

/* Source: ssygst.f */
#define ssygst FORTRAN_WRAPPER(ssygst)
extern void ssygst(
    ptrdiff_t *itype,
    char   *uplo,
    ptrdiff_t *n,
    float  *a,
    ptrdiff_t *lda,
    float  *b,
    ptrdiff_t *ldb,
    ptrdiff_t *info
);

/* Source: ssygv.f */
#define ssygv FORTRAN_WRAPPER(ssygv)
extern void ssygv(
    ptrdiff_t *itype,
    char   *jobz,
    char   *uplo,
    ptrdiff_t *n,
    float  *a,
    ptrdiff_t *lda,
    float  *b,
    ptrdiff_t *ldb,
    float  *w,
    float  *work,
    ptrdiff_t *lwork,
    ptrdiff_t *info
);

/* Source: ssygvd.f */
#define ssygvd FORTRAN_WRAPPER(ssygvd)
extern void ssygvd(
    ptrdiff_t *itype,
    char   *jobz,
    char   *uplo,
    ptrdiff_t *n,
    float  *a,
    ptrdiff_t *lda,
    float  *b,
    ptrdiff_t *ldb,
    float  *w,
    float  *work,
    ptrdiff_t *lwork,
    ptrdiff_t *iwork,
    ptrdiff_t *liwork,
    ptrdiff_t *info
);

/* Source: ssygvx.f */
#define ssygvx FORTRAN_WRAPPER(ssygvx)
extern void ssygvx(
    ptrdiff_t *itype,
    char   *jobz,
    char   *range,
    char   *uplo,
    ptrdiff_t *n,
    float  *a,
    ptrdiff_t *lda,
    float  *b,
    ptrdiff_t *ldb,
    float  *vl,
    float  *vu,
    ptrdiff_t *il,
    ptrdiff_t *iu,
    float  *abstol,
    ptrdiff_t *m,
    float  *w,
    float  *z,
    ptrdiff_t *ldz,
    float  *work,
    ptrdiff_t *lwork,
    ptrdiff_t *iwork,
    ptrdiff_t *ifail,
    ptrdiff_t *info
);

/* Source: ssyrfs.f */
#define ssyrfs FORTRAN_WRAPPER(ssyrfs)
extern void ssyrfs(
    char   *uplo,
    ptrdiff_t *n,
    ptrdiff_t *nrhs,
    float  *a,
    ptrdiff_t *lda,
    float  *af,
    ptrdiff_t *ldaf,
    ptrdiff_t *ipiv,
    float  *b,
    ptrdiff_t *ldb,
    float  *x,
    ptrdiff_t *ldx,
    float  *ferr,
    float  *berr,
    float  *work,
    ptrdiff_t *iwork,
    ptrdiff_t *info
);

/* Source: ssysv.f */
#define ssysv FORTRAN_WRAPPER(ssysv)
extern void ssysv(
    char   *uplo,
    ptrdiff_t *n,
    ptrdiff_t *nrhs,
    float  *a,
    ptrdiff_t *lda,
    ptrdiff_t *ipiv,
    float  *b,
    ptrdiff_t *ldb,
    float  *work,
    ptrdiff_t *lwork,
    ptrdiff_t *info
);

/* Source: ssysvx.f */
#define ssysvx FORTRAN_WRAPPER(ssysvx)
extern void ssysvx(
    char   *fact,
    char   *uplo,
    ptrdiff_t *n,
    ptrdiff_t *nrhs,
    float  *a,
    ptrdiff_t *lda,
    float  *af,
    ptrdiff_t *ldaf,
    ptrdiff_t *ipiv,
    float  *b,
    ptrdiff_t *ldb,
    float  *x,
    ptrdiff_t *ldx,
    float  *rcond,
    float  *ferr,
    float  *berr,
    float  *work,
    ptrdiff_t *lwork,
    ptrdiff_t *iwork,
    ptrdiff_t *info
);

/* Source: ssytd2.f */
#define ssytd2 FORTRAN_WRAPPER(ssytd2)
extern void ssytd2(
    char   *uplo,
    ptrdiff_t *n,
    float  *a,
    ptrdiff_t *lda,
    float  *d,
    float  *e,
    float  *tau,
    ptrdiff_t *info
);

/* Source: ssytf2.f */
#define ssytf2 FORTRAN_WRAPPER(ssytf2)
extern void ssytf2(
    char   *uplo,
    ptrdiff_t *n,
    float  *a,
    ptrdiff_t *lda,
    ptrdiff_t *ipiv,
    ptrdiff_t *info
);

/* Source: ssytrd.f */
#define ssytrd FORTRAN_WRAPPER(ssytrd)
extern void ssytrd(
    char   *uplo,
    ptrdiff_t *n,
    float  *a,
    ptrdiff_t *lda,
    float  *d,
    float  *e,
    float  *tau,
    float  *work,
    ptrdiff_t *lwork,
    ptrdiff_t *info
);

/* Source: ssytrf.f */
#define ssytrf FORTRAN_WRAPPER(ssytrf)
extern void ssytrf(
    char   *uplo,
    ptrdiff_t *n,
    float  *a,
    ptrdiff_t *lda,
    ptrdiff_t *ipiv,
    float  *work,
    ptrdiff_t *lwork,
    ptrdiff_t *info
);

/* Source: ssytri.f */
#define ssytri FORTRAN_WRAPPER(ssytri)
extern void ssytri(
    char   *uplo,
    ptrdiff_t *n,
    float  *a,
    ptrdiff_t *lda,
    ptrdiff_t *ipiv,
    float  *work,
    ptrdiff_t *info
);

/* Source: ssytrs.f */
#define ssytrs FORTRAN_WRAPPER(ssytrs)
extern void ssytrs(
    char   *uplo,
    ptrdiff_t *n,
    ptrdiff_t *nrhs,
    float  *a,
    ptrdiff_t *lda,
    ptrdiff_t *ipiv,
    float  *b,
    ptrdiff_t *ldb,
    ptrdiff_t *info
);

/* Source: stbcon.f */
#define stbcon FORTRAN_WRAPPER(stbcon)
extern void stbcon(
    char   *norm,
    char   *uplo,
    char   *diag,
    ptrdiff_t *n,
    ptrdiff_t *kd,
    float  *ab,
    ptrdiff_t *ldab,
    float  *rcond,
    float  *work,
    ptrdiff_t *iwork,
    ptrdiff_t *info
);

/* Source: stbrfs.f */
#define stbrfs FORTRAN_WRAPPER(stbrfs)
extern void stbrfs(
    char   *uplo,
    char   *trans,
    char   *diag,
    ptrdiff_t *n,
    ptrdiff_t *kd,
    ptrdiff_t *nrhs,
    float  *ab,
    ptrdiff_t *ldab,
    float  *b,
    ptrdiff_t *ldb,
    float  *x,
    ptrdiff_t *ldx,
    float  *ferr,
    float  *berr,
    float  *work,
    ptrdiff_t *iwork,
    ptrdiff_t *info
);

/* Source: stbtrs.f */
#define stbtrs FORTRAN_WRAPPER(stbtrs)
extern void stbtrs(
    char   *uplo,
    char   *trans,
    char   *diag,
    ptrdiff_t *n,
    ptrdiff_t *kd,
    ptrdiff_t *nrhs,
    float  *ab,
    ptrdiff_t *ldab,
    float  *b,
    ptrdiff_t *ldb,
    ptrdiff_t *info
);

/* Source: stfsm.f */
#define stfsm FORTRAN_WRAPPER(stfsm)
extern void stfsm(
    char   *transr,
    char   *side,
    char   *uplo,
    char   *trans,
    char   *diag,
    ptrdiff_t *m,
    ptrdiff_t *n,
    float  *alpha,
    float  *a,
    float  *b,
    ptrdiff_t *ldb
);

/* Source: stftri.f */
#define stftri FORTRAN_WRAPPER(stftri)
extern void stftri(
    char   *transr,
    char   *uplo,
    char   *diag,
    ptrdiff_t *n,
    float  *a,
    ptrdiff_t *info
);

/* Source: stfttp.f */
#define stfttp FORTRAN_WRAPPER(stfttp)
extern void stfttp(
    char   *transr,
    char   *uplo,
    ptrdiff_t *n,
    float  *arf,
    float  *ap,
    ptrdiff_t *info
);

/* Source: stfttr.f */
#define stfttr FORTRAN_WRAPPER(stfttr)
extern void stfttr(
    char   *transr,
    char   *uplo,
    ptrdiff_t *n,
    float  *arf,
    float  *a,
    ptrdiff_t *lda,
    ptrdiff_t *info
);

/* Source: stgevc.f */
#define stgevc FORTRAN_WRAPPER(stgevc)
extern void stgevc(
    char   *side,
    char   *howmny,
    ptrdiff_t *select,
    ptrdiff_t *n,
    float  *s,
    ptrdiff_t *lds,
    float  *p,
    ptrdiff_t *ldp,
    float  *vl,
    ptrdiff_t *ldvl,
    float  *vr,
    ptrdiff_t *ldvr,
    ptrdiff_t *mm,
    ptrdiff_t *m,
    float  *work,
    ptrdiff_t *info
);

/* Source: stgex2.f */
#define stgex2 FORTRAN_WRAPPER(stgex2)
extern void stgex2(
    ptrdiff_t *wantq,
    ptrdiff_t *wantz,
    ptrdiff_t *n,
    float  *a,
    ptrdiff_t *lda,
    float  *b,
    ptrdiff_t *ldb,
    float  *q,
    ptrdiff_t *ldq,
    float  *z,
    ptrdiff_t *ldz,
    ptrdiff_t *j1_,
    ptrdiff_t *n1,
    ptrdiff_t *n2,
    float  *work,
    ptrdiff_t *lwork,
    ptrdiff_t *info
);

/* Source: stgexc.f */
#define stgexc FORTRAN_WRAPPER(stgexc)
extern void stgexc(
    ptrdiff_t *wantq,
    ptrdiff_t *wantz,
    ptrdiff_t *n,
    float  *a,
    ptrdiff_t *lda,
    float  *b,
    ptrdiff_t *ldb,
    float  *q,
    ptrdiff_t *ldq,
    float  *z,
    ptrdiff_t *ldz,
    ptrdiff_t *ifst,
    ptrdiff_t *ilst,
    float  *work,
    ptrdiff_t *lwork,
    ptrdiff_t *info
);

/* Source: stgsen.f */
#define stgsen FORTRAN_WRAPPER(stgsen)
extern void stgsen(
    ptrdiff_t *ijob,
    ptrdiff_t *wantq,
    ptrdiff_t *wantz,
    ptrdiff_t *select,
    ptrdiff_t *n,
    float  *a,
    ptrdiff_t *lda,
    float  *b,
    ptrdiff_t *ldb,
    float  *alphar,
    float  *alphai,
    float  *beta,
    float  *q,
    ptrdiff_t *ldq,
    float  *z,
    ptrdiff_t *ldz,
    ptrdiff_t *m,
    float  *pl,
    float  *pr,
    float  *dif,
    float  *work,
    ptrdiff_t *lwork,
    ptrdiff_t *iwork,
    ptrdiff_t *liwork,
    ptrdiff_t *info
);

/* Source: stgsja.f */
#define stgsja FORTRAN_WRAPPER(stgsja)
extern void stgsja(
    char   *jobu,
    char   *jobv,
    char   *jobq,
    ptrdiff_t *m,
    ptrdiff_t *p,
    ptrdiff_t *n,
    ptrdiff_t *k,
    ptrdiff_t *l,
    float  *a,
    ptrdiff_t *lda,
    float  *b,
    ptrdiff_t *ldb,
    float  *tola,
    float  *tolb,
    float  *alpha,
    float  *beta,
    float  *u,
    ptrdiff_t *ldu,
    float  *v,
    ptrdiff_t *ldv,
    float  *q,
    ptrdiff_t *ldq,
    float  *work,
    ptrdiff_t *ncycle,
    ptrdiff_t *info
);

/* Source: stgsna.f */
#define stgsna FORTRAN_WRAPPER(stgsna)
extern void stgsna(
    char   *job,
    char   *howmny,
    ptrdiff_t *select,
    ptrdiff_t *n,
    float  *a,
    ptrdiff_t *lda,
    float  *b,
    ptrdiff_t *ldb,
    float  *vl,
    ptrdiff_t *ldvl,
    float  *vr,
    ptrdiff_t *ldvr,
    float  *s,
    float  *dif,
    ptrdiff_t *mm,
    ptrdiff_t *m,
    float  *work,
    ptrdiff_t *lwork,
    ptrdiff_t *iwork,
    ptrdiff_t *info
);

/* Source: stgsy2.f */
#define stgsy2 FORTRAN_WRAPPER(stgsy2)
extern void stgsy2(
    char   *trans,
    ptrdiff_t *ijob,
    ptrdiff_t *m,
    ptrdiff_t *n,
    float  *a,
    ptrdiff_t *lda,
    float  *b,
    ptrdiff_t *ldb,
    float  *c,
    ptrdiff_t *ldc,
    float  *d,
    ptrdiff_t *ldd,
    float  *e,
    ptrdiff_t *lde,
    float  *f,
    ptrdiff_t *ldf,
    float  *scale,
    float  *rdsum,
    float  *rdscal,
    ptrdiff_t *iwork,
    ptrdiff_t *pq,
    ptrdiff_t *info
);

/* Source: stgsyl.f */
#define stgsyl FORTRAN_WRAPPER(stgsyl)
extern void stgsyl(
    char   *trans,
    ptrdiff_t *ijob,
    ptrdiff_t *m,
    ptrdiff_t *n,
    float  *a,
    ptrdiff_t *lda,
    float  *b,
    ptrdiff_t *ldb,
    float  *c,
    ptrdiff_t *ldc,
    float  *d,
    ptrdiff_t *ldd,
    float  *e,
    ptrdiff_t *lde,
    float  *f,
    ptrdiff_t *ldf,
    float  *scale,
    float  *dif,
    float  *work,
    ptrdiff_t *lwork,
    ptrdiff_t *iwork,
    ptrdiff_t *info
);

/* Source: stpcon.f */
#define stpcon FORTRAN_WRAPPER(stpcon)
extern void stpcon(
    char   *norm,
    char   *uplo,
    char   *diag,
    ptrdiff_t *n,
    float  *ap,
    float  *rcond,
    float  *work,
    ptrdiff_t *iwork,
    ptrdiff_t *info
);

/* Source: stprfs.f */
#define stprfs FORTRAN_WRAPPER(stprfs)
extern void stprfs(
    char   *uplo,
    char   *trans,
    char   *diag,
    ptrdiff_t *n,
    ptrdiff_t *nrhs,
    float  *ap,
    float  *b,
    ptrdiff_t *ldb,
    float  *x,
    ptrdiff_t *ldx,
    float  *ferr,
    float  *berr,
    float  *work,
    ptrdiff_t *iwork,
    ptrdiff_t *info
);

/* Source: stptri.f */
#define stptri FORTRAN_WRAPPER(stptri)
extern void stptri(
    char   *uplo,
    char   *diag,
    ptrdiff_t *n,
    float  *ap,
    ptrdiff_t *info
);

/* Source: stptrs.f */
#define stptrs FORTRAN_WRAPPER(stptrs)
extern void stptrs(
    char   *uplo,
    char   *trans,
    char   *diag,
    ptrdiff_t *n,
    ptrdiff_t *nrhs,
    float  *ap,
    float  *b,
    ptrdiff_t *ldb,
    ptrdiff_t *info
);

/* Source: stpttf.f */
#define stpttf FORTRAN_WRAPPER(stpttf)
extern void stpttf(
    char   *transr,
    char   *uplo,
    ptrdiff_t *n,
    float  *ap,
    float  *arf,
    ptrdiff_t *info
);

/* Source: stpttr.f */
#define stpttr FORTRAN_WRAPPER(stpttr)
extern void stpttr(
    char   *uplo,
    ptrdiff_t *n,
    float  *ap,
    float  *a,
    ptrdiff_t *lda,
    ptrdiff_t *info
);

/* Source: strcon.f */
#define strcon FORTRAN_WRAPPER(strcon)
extern void strcon(
    char   *norm,
    char   *uplo,
    char   *diag,
    ptrdiff_t *n,
    float  *a,
    ptrdiff_t *lda,
    float  *rcond,
    float  *work,
    ptrdiff_t *iwork,
    ptrdiff_t *info
);

/* Source: strevc.f */
#define strevc FORTRAN_WRAPPER(strevc)
extern void strevc(
    char   *side,
    char   *howmny,
    ptrdiff_t *select,
    ptrdiff_t *n,
    float  *t,
    ptrdiff_t *ldt,
    float  *vl,
    ptrdiff_t *ldvl,
    float  *vr,
    ptrdiff_t *ldvr,
    ptrdiff_t *mm,
    ptrdiff_t *m,
    float  *work,
    ptrdiff_t *info
);

/* Source: strexc.f */
#define strexc FORTRAN_WRAPPER(strexc)
extern void strexc(
    char   *compq,
    ptrdiff_t *n,
    float  *t,
    ptrdiff_t *ldt,
    float  *q,
    ptrdiff_t *ldq,
    ptrdiff_t *ifst,
    ptrdiff_t *ilst,
    float  *work,
    ptrdiff_t *info
);

/* Source: strrfs.f */
#define strrfs FORTRAN_WRAPPER(strrfs)
extern void strrfs(
    char   *uplo,
    char   *trans,
    char   *diag,
    ptrdiff_t *n,
    ptrdiff_t *nrhs,
    float  *a,
    ptrdiff_t *lda,
    float  *b,
    ptrdiff_t *ldb,
    float  *x,
    ptrdiff_t *ldx,
    float  *ferr,
    float  *berr,
    float  *work,
    ptrdiff_t *iwork,
    ptrdiff_t *info
);

/* Source: strsen.f */
#define strsen FORTRAN_WRAPPER(strsen)
extern void strsen(
    char   *job,
    char   *compq,
    ptrdiff_t *select,
    ptrdiff_t *n,
    float  *t,
    ptrdiff_t *ldt,
    float  *q,
    ptrdiff_t *ldq,
    float  *wr,
    float  *wi,
    ptrdiff_t *m,
    float  *s,
    float  *sep,
    float  *work,
    ptrdiff_t *lwork,
    ptrdiff_t *iwork,
    ptrdiff_t *liwork,
    ptrdiff_t *info
);

/* Source: strsna.f */
#define strsna FORTRAN_WRAPPER(strsna)
extern void strsna(
    char   *job,
    char   *howmny,
    ptrdiff_t *select,
    ptrdiff_t *n,
    float  *t,
    ptrdiff_t *ldt,
    float  *vl,
    ptrdiff_t *ldvl,
    float  *vr,
    ptrdiff_t *ldvr,
    float  *s,
    float  *sep,
    ptrdiff_t *mm,
    ptrdiff_t *m,
    float  *work,
    ptrdiff_t *ldwork,
    ptrdiff_t *iwork,
    ptrdiff_t *info
);

/* Source: strsyl.f */
#define strsyl FORTRAN_WRAPPER(strsyl)
extern void strsyl(
    char   *trana,
    char   *tranb,
    ptrdiff_t *isgn,
    ptrdiff_t *m,
    ptrdiff_t *n,
    float  *a,
    ptrdiff_t *lda,
    float  *b,
    ptrdiff_t *ldb,
    float  *c,
    ptrdiff_t *ldc,
    float  *scale,
    ptrdiff_t *info
);

/* Source: strti2.f */
#define strti2 FORTRAN_WRAPPER(strti2)
extern void strti2(
    char   *uplo,
    char   *diag,
    ptrdiff_t *n,
    float  *a,
    ptrdiff_t *lda,
    ptrdiff_t *info
);

/* Source: strtri.f */
#define strtri FORTRAN_WRAPPER(strtri)
extern void strtri(
    char   *uplo,
    char   *diag,
    ptrdiff_t *n,
    float  *a,
    ptrdiff_t *lda,
    ptrdiff_t *info
);

/* Source: strtrs.f */
#define strtrs FORTRAN_WRAPPER(strtrs)
extern void strtrs(
    char   *uplo,
    char   *trans,
    char   *diag,
    ptrdiff_t *n,
    ptrdiff_t *nrhs,
    float  *a,
    ptrdiff_t *lda,
    float  *b,
    ptrdiff_t *ldb,
    ptrdiff_t *info
);

/* Source: strttf.f */
#define strttf FORTRAN_WRAPPER(strttf)
extern void strttf(
    char   *transr,
    char   *uplo,
    ptrdiff_t *n,
    float  *a,
    ptrdiff_t *lda,
    float  *arf,
    ptrdiff_t *info
);

/* Source: strttp.f */
#define strttp FORTRAN_WRAPPER(strttp)
extern void strttp(
    char   *uplo,
    ptrdiff_t *n,
    float  *a,
    ptrdiff_t *lda,
    float  *ap,
    ptrdiff_t *info
);

/* Source: stzrqf.f */
#define stzrqf FORTRAN_WRAPPER(stzrqf)
extern void stzrqf(
    ptrdiff_t *m,
    ptrdiff_t *n,
    float  *a,
    ptrdiff_t *lda,
    float  *tau,
    ptrdiff_t *info
);

/* Source: stzrzf.f */
#define stzrzf FORTRAN_WRAPPER(stzrzf)
extern void stzrzf(
    ptrdiff_t *m,
    ptrdiff_t *n,
    float  *a,
    ptrdiff_t *lda,
    float  *tau,
    float  *work,
    ptrdiff_t *lwork,
    ptrdiff_t *info
);

/* Source: xerbla_array.f */
#define xerbla_array FORTRAN_WRAPPER(xerbla_array)
extern void xerbla_array(
    char   *srname_array,
    ptrdiff_t *srname_len,
    ptrdiff_t *info
);

/* Source: zbdsqr.f */
#define zbdsqr FORTRAN_WRAPPER(zbdsqr)
extern void zbdsqr(
    char   *uplo,
    ptrdiff_t *n,
    ptrdiff_t *ncvt,
    ptrdiff_t *nru,
    ptrdiff_t *ncc,
    double *d,
    double *e,
    double *vt,
    ptrdiff_t *ldvt,
    double *u,
    ptrdiff_t *ldu,
    double *c,
    ptrdiff_t *ldc,
    double *rwork,
    ptrdiff_t *info
);

/* Source: zcgesv.f */
#define zcgesv FORTRAN_WRAPPER(zcgesv)
extern void zcgesv(
    ptrdiff_t *n,
    ptrdiff_t *nrhs,
    double *a,
    ptrdiff_t *lda,
    ptrdiff_t *ipiv,
    double *b,
    ptrdiff_t *ldb,
    double *x,
    ptrdiff_t *ldx,
    double *work,
    float  *swork,
    double *rwork,
    ptrdiff_t *iter,
    ptrdiff_t *info
);

/* Source: zcposv.f */
#define zcposv FORTRAN_WRAPPER(zcposv)
extern void zcposv(
    char   *uplo,
    ptrdiff_t *n,
    ptrdiff_t *nrhs,
    double *a,
    ptrdiff_t *lda,
    double *b,
    ptrdiff_t *ldb,
    double *x,
    ptrdiff_t *ldx,
    double *work,
    float  *swork,
    double *rwork,
    ptrdiff_t *iter,
    ptrdiff_t *info
);

/* Source: zdrscl.f */
#define zdrscl FORTRAN_WRAPPER(zdrscl)
extern void zdrscl(
    ptrdiff_t *n,
    double *sa,
    double *sx,
    ptrdiff_t *incx
);

/* Source: zgbbrd.f */
#define zgbbrd FORTRAN_WRAPPER(zgbbrd)
extern void zgbbrd(
    char   *vect,
    ptrdiff_t *m,
    ptrdiff_t *n,
    ptrdiff_t *ncc,
    ptrdiff_t *kl,
    ptrdiff_t *ku,
    double *ab,
    ptrdiff_t *ldab,
    double *d,
    double *e,
    double *q,
    ptrdiff_t *ldq,
    double *pt,
    ptrdiff_t *ldpt,
    double *c,
    ptrdiff_t *ldc,
    double *work,
    double *rwork,
    ptrdiff_t *info
);

/* Source: zgbcon.f */
#define zgbcon FORTRAN_WRAPPER(zgbcon)
extern void zgbcon(
    char   *norm,
    ptrdiff_t *n,
    ptrdiff_t *kl,
    ptrdiff_t *ku,
    double *ab,
    ptrdiff_t *ldab,
    ptrdiff_t *ipiv,
    double *anorm,
    double *rcond,
    double *work,
    double *rwork,
    ptrdiff_t *info
);

/* Source: zgbequ.f */
#define zgbequ FORTRAN_WRAPPER(zgbequ)
extern void zgbequ(
    ptrdiff_t *m,
    ptrdiff_t *n,
    ptrdiff_t *kl,
    ptrdiff_t *ku,
    double *ab,
    ptrdiff_t *ldab,
    double *r,
    double *c,
    double *rowcnd,
    double *colcnd,
    double *amax,
    ptrdiff_t *info
);

/* Source: zgbequb.f */
#define zgbequb FORTRAN_WRAPPER(zgbequb)
extern void zgbequb(
    ptrdiff_t *m,
    ptrdiff_t *n,
    ptrdiff_t *kl,
    ptrdiff_t *ku,
    double *ab,
    ptrdiff_t *ldab,
    double *r,
    double *c,
    double *rowcnd,
    double *colcnd,
    double *amax,
    ptrdiff_t *info
);

/* Source: zgbrfs.f */
#define zgbrfs FORTRAN_WRAPPER(zgbrfs)
extern void zgbrfs(
    char   *trans,
    ptrdiff_t *n,
    ptrdiff_t *kl,
    ptrdiff_t *ku,
    ptrdiff_t *nrhs,
    double *ab,
    ptrdiff_t *ldab,
    double *afb,
    ptrdiff_t *ldafb,
    ptrdiff_t *ipiv,
    double *b,
    ptrdiff_t *ldb,
    double *x,
    ptrdiff_t *ldx,
    double *ferr,
    double *berr,
    double *work,
    double *rwork,
    ptrdiff_t *info
);

/* Source: zgbsv.f */
#define zgbsv FORTRAN_WRAPPER(zgbsv)
extern void zgbsv(
    ptrdiff_t *n,
    ptrdiff_t *kl,
    ptrdiff_t *ku,
    ptrdiff_t *nrhs,
    double *ab,
    ptrdiff_t *ldab,
    ptrdiff_t *ipiv,
    double *b,
    ptrdiff_t *ldb,
    ptrdiff_t *info
);

/* Source: zgbsvx.f */
#define zgbsvx FORTRAN_WRAPPER(zgbsvx)
extern void zgbsvx(
    char   *fact,
    char   *trans,
    ptrdiff_t *n,
    ptrdiff_t *kl,
    ptrdiff_t *ku,
    ptrdiff_t *nrhs,
    double *ab,
    ptrdiff_t *ldab,
    double *afb,
    ptrdiff_t *ldafb,
    ptrdiff_t *ipiv,
    char   *equed,
    double *r,
    double *c,
    double *b,
    ptrdiff_t *ldb,
    double *x,
    ptrdiff_t *ldx,
    double *rcond,
    double *ferr,
    double *berr,
    double *work,
    double *rwork,
    ptrdiff_t *info
);

/* Source: zgbtf2.f */
#define zgbtf2 FORTRAN_WRAPPER(zgbtf2)
extern void zgbtf2(
    ptrdiff_t *m,
    ptrdiff_t *n,
    ptrdiff_t *kl,
    ptrdiff_t *ku,
    double *ab,
    ptrdiff_t *ldab,
    ptrdiff_t *ipiv,
    ptrdiff_t *info
);

/* Source: zgbtrf.f */
#define zgbtrf FORTRAN_WRAPPER(zgbtrf)
extern void zgbtrf(
    ptrdiff_t *m,
    ptrdiff_t *n,
    ptrdiff_t *kl,
    ptrdiff_t *ku,
    double *ab,
    ptrdiff_t *ldab,
    ptrdiff_t *ipiv,
    ptrdiff_t *info
);

/* Source: zgbtrs.f */
#define zgbtrs FORTRAN_WRAPPER(zgbtrs)
extern void zgbtrs(
    char   *trans,
    ptrdiff_t *n,
    ptrdiff_t *kl,
    ptrdiff_t *ku,
    ptrdiff_t *nrhs,
    double *ab,
    ptrdiff_t *ldab,
    ptrdiff_t *ipiv,
    double *b,
    ptrdiff_t *ldb,
    ptrdiff_t *info
);

/* Source: zgebak.f */
#define zgebak FORTRAN_WRAPPER(zgebak)
extern void zgebak(
    char   *job,
    char   *side,
    ptrdiff_t *n,
    ptrdiff_t *ilo,
    ptrdiff_t *ihi,
    double *scale,
    ptrdiff_t *m,
    double *v,
    ptrdiff_t *ldv,
    ptrdiff_t *info
);

/* Source: zgebal.f */
#define zgebal FORTRAN_WRAPPER(zgebal)
extern void zgebal(
    char   *job,
    ptrdiff_t *n,
    double *a,
    ptrdiff_t *lda,
    ptrdiff_t *ilo,
    ptrdiff_t *ihi,
    double *scale,
    ptrdiff_t *info
);

/* Source: zgebd2.f */
#define zgebd2 FORTRAN_WRAPPER(zgebd2)
extern void zgebd2(
    ptrdiff_t *m,
    ptrdiff_t *n,
    double *a,
    ptrdiff_t *lda,
    double *d,
    double *e,
    double *tauq,
    double *taup,
    double *work,
    ptrdiff_t *info
);

/* Source: zgebrd.f */
#define zgebrd FORTRAN_WRAPPER(zgebrd)
extern void zgebrd(
    ptrdiff_t *m,
    ptrdiff_t *n,
    double *a,
    ptrdiff_t *lda,
    double *d,
    double *e,
    double *tauq,
    double *taup,
    double *work,
    ptrdiff_t *lwork,
    ptrdiff_t *info
);

/* Source: zgecon.f */
#define zgecon FORTRAN_WRAPPER(zgecon)
extern void zgecon(
    char   *norm,
    ptrdiff_t *n,
    double *a,
    ptrdiff_t *lda,
    double *anorm,
    double *rcond,
    double *work,
    double *rwork,
    ptrdiff_t *info
);

/* Source: zgeequ.f */
#define zgeequ FORTRAN_WRAPPER(zgeequ)
extern void zgeequ(
    ptrdiff_t *m,
    ptrdiff_t *n,
    double *a,
    ptrdiff_t *lda,
    double *r,
    double *c,
    double *rowcnd,
    double *colcnd,
    double *amax,
    ptrdiff_t *info
);

/* Source: zgeequb.f */
#define zgeequb FORTRAN_WRAPPER(zgeequb)
extern void zgeequb(
    ptrdiff_t *m,
    ptrdiff_t *n,
    double *a,
    ptrdiff_t *lda,
    double *r,
    double *c,
    double *rowcnd,
    double *colcnd,
    double *amax,
    ptrdiff_t *info
);

/* Source: zgees.f */
#define zgees FORTRAN_WRAPPER(zgees)
extern void zgees(
    char   *jobvs,
    char   *sort,
    ptrdiff_t (*select)(),
    ptrdiff_t *n,
    double *a,
    ptrdiff_t *lda,
    ptrdiff_t *sdim,
    double *w,
    double *vs,
    ptrdiff_t *ldvs,
    double *work,
    ptrdiff_t *lwork,
    double *rwork,
    ptrdiff_t *bwork,
    ptrdiff_t *info
);

/* Source: zgeesx.f */
#define zgeesx FORTRAN_WRAPPER(zgeesx)
extern void zgeesx(
    char   *jobvs,
    char   *sort,
    ptrdiff_t (*select)(),
    char   *sense,
    ptrdiff_t *n,
    double *a,
    ptrdiff_t *lda,
    ptrdiff_t *sdim,
    double *w,
    double *vs,
    ptrdiff_t *ldvs,
    double *rconde,
    double *rcondv,
    double *work,
    ptrdiff_t *lwork,
    double *rwork,
    ptrdiff_t *bwork,
    ptrdiff_t *info
);

/* Source: zgeev.f */
#define zgeev FORTRAN_WRAPPER(zgeev)
extern void zgeev(
    char   *jobvl,
    char   *jobvr,
    ptrdiff_t *n,
    double *a,
    ptrdiff_t *lda,
    double *w,
    double *vl,
    ptrdiff_t *ldvl,
    double *vr,
    ptrdiff_t *ldvr,
    double *work,
    ptrdiff_t *lwork,
    double *rwork,
    ptrdiff_t *info
);

/* Source: zgeevx.f */
#define zgeevx FORTRAN_WRAPPER(zgeevx)
extern void zgeevx(
    char   *balanc,
    char   *jobvl,
    char   *jobvr,
    char   *sense,
    ptrdiff_t *n,
    double *a,
    ptrdiff_t *lda,
    double *w,
    double *vl,
    ptrdiff_t *ldvl,
    double *vr,
    ptrdiff_t *ldvr,
    ptrdiff_t *ilo,
    ptrdiff_t *ihi,
    double *scale,
    double *abnrm,
    double *rconde,
    double *rcondv,
    double *work,
    ptrdiff_t *lwork,
    double *rwork,
    ptrdiff_t *info
);

/* Source: zgegs.f */
#define zgegs FORTRAN_WRAPPER(zgegs)
extern void zgegs(
    char   *jobvsl,
    char   *jobvsr,
    ptrdiff_t *n,
    double *a,
    ptrdiff_t *lda,
    double *b,
    ptrdiff_t *ldb,
    double *alpha,
    double *beta,
    double *vsl,
    ptrdiff_t *ldvsl,
    double *vsr,
    ptrdiff_t *ldvsr,
    double *work,
    ptrdiff_t *lwork,
    double *rwork,
    ptrdiff_t *info
);

/* Source: zgegv.f */
#define zgegv FORTRAN_WRAPPER(zgegv)
extern void zgegv(
    char   *jobvl,
    char   *jobvr,
    ptrdiff_t *n,
    double *a,
    ptrdiff_t *lda,
    double *b,
    ptrdiff_t *ldb,
    double *alpha,
    double *beta,
    double *vl,
    ptrdiff_t *ldvl,
    double *vr,
    ptrdiff_t *ldvr,
    double *work,
    ptrdiff_t *lwork,
    double *rwork,
    ptrdiff_t *info
);

/* Source: zgehd2.f */
#define zgehd2 FORTRAN_WRAPPER(zgehd2)
extern void zgehd2(
    ptrdiff_t *n,
    ptrdiff_t *ilo,
    ptrdiff_t *ihi,
    double *a,
    ptrdiff_t *lda,
    double *tau,
    double *work,
    ptrdiff_t *info
);

/* Source: zgehrd.f */
#define zgehrd FORTRAN_WRAPPER(zgehrd)
extern void zgehrd(
    ptrdiff_t *n,
    ptrdiff_t *ilo,
    ptrdiff_t *ihi,
    double *a,
    ptrdiff_t *lda,
    double *tau,
    double *work,
    ptrdiff_t *lwork,
    ptrdiff_t *info
);

/* Source: zgelq2.f */
#define zgelq2 FORTRAN_WRAPPER(zgelq2)
extern void zgelq2(
    ptrdiff_t *m,
    ptrdiff_t *n,
    double *a,
    ptrdiff_t *lda,
    double *tau,
    double *work,
    ptrdiff_t *info
);

/* Source: zgelqf.f */
#define zgelqf FORTRAN_WRAPPER(zgelqf)
extern void zgelqf(
    ptrdiff_t *m,
    ptrdiff_t *n,
    double *a,
    ptrdiff_t *lda,
    double *tau,
    double *work,
    ptrdiff_t *lwork,
    ptrdiff_t *info
);

/* Source: zgels.f */
#define zgels FORTRAN_WRAPPER(zgels)
extern void zgels(
    char   *trans,
    ptrdiff_t *m,
    ptrdiff_t *n,
    ptrdiff_t *nrhs,
    double *a,
    ptrdiff_t *lda,
    double *b,
    ptrdiff_t *ldb,
    double *work,
    ptrdiff_t *lwork,
    ptrdiff_t *info
);

/* Source: zgelsd.f */
#define zgelsd FORTRAN_WRAPPER(zgelsd)
extern void zgelsd(
    ptrdiff_t *m,
    ptrdiff_t *n,
    ptrdiff_t *nrhs,
    double *a,
    ptrdiff_t *lda,
    double *b,
    ptrdiff_t *ldb,
    double *s,
    double *rcond,
    ptrdiff_t *rank,
    double *work,
    ptrdiff_t *lwork,
    double *rwork,
    ptrdiff_t *iwork,
    ptrdiff_t *info
);

/* Source: zgelss.f */
#define zgelss FORTRAN_WRAPPER(zgelss)
extern void zgelss(
    ptrdiff_t *m,
    ptrdiff_t *n,
    ptrdiff_t *nrhs,
    double *a,
    ptrdiff_t *lda,
    double *b,
    ptrdiff_t *ldb,
    double *s,
    double *rcond,
    ptrdiff_t *rank,
    double *work,
    ptrdiff_t *lwork,
    double *rwork,
    ptrdiff_t *info
);

/* Source: zgelsx.f */
#define zgelsx FORTRAN_WRAPPER(zgelsx)
extern void zgelsx(
    ptrdiff_t *m,
    ptrdiff_t *n,
    ptrdiff_t *nrhs,
    double *a,
    ptrdiff_t *lda,
    double *b,
    ptrdiff_t *ldb,
    ptrdiff_t *jpvt,
    double *rcond,
    ptrdiff_t *rank,
    double *work,
    double *rwork,
    ptrdiff_t *info
);

/* Source: zgelsy.f */
#define zgelsy FORTRAN_WRAPPER(zgelsy)
extern void zgelsy(
    ptrdiff_t *m,
    ptrdiff_t *n,
    ptrdiff_t *nrhs,
    double *a,
    ptrdiff_t *lda,
    double *b,
    ptrdiff_t *ldb,
    ptrdiff_t *jpvt,
    double *rcond,
    ptrdiff_t *rank,
    double *work,
    ptrdiff_t *lwork,
    double *rwork,
    ptrdiff_t *info
);

/* Source: zgeql2.f */
#define zgeql2 FORTRAN_WRAPPER(zgeql2)
extern void zgeql2(
    ptrdiff_t *m,
    ptrdiff_t *n,
    double *a,
    ptrdiff_t *lda,
    double *tau,
    double *work,
    ptrdiff_t *info
);

/* Source: zgeqlf.f */
#define zgeqlf FORTRAN_WRAPPER(zgeqlf)
extern void zgeqlf(
    ptrdiff_t *m,
    ptrdiff_t *n,
    double *a,
    ptrdiff_t *lda,
    double *tau,
    double *work,
    ptrdiff_t *lwork,
    ptrdiff_t *info
);

/* Source: zgeqp3.f */
#define zgeqp3 FORTRAN_WRAPPER(zgeqp3)
extern void zgeqp3(
    ptrdiff_t *m,
    ptrdiff_t *n,
    double *a,
    ptrdiff_t *lda,
    ptrdiff_t *jpvt,
    double *tau,
    double *work,
    ptrdiff_t *lwork,
    double *rwork,
    ptrdiff_t *info
);

/* Source: zgeqpf.f */
#define zgeqpf FORTRAN_WRAPPER(zgeqpf)
extern void zgeqpf(
    ptrdiff_t *m,
    ptrdiff_t *n,
    double *a,
    ptrdiff_t *lda,
    ptrdiff_t *jpvt,
    double *tau,
    double *work,
    double *rwork,
    ptrdiff_t *info
);

/* Source: zgeqr2.f */
#define zgeqr2 FORTRAN_WRAPPER(zgeqr2)
extern void zgeqr2(
    ptrdiff_t *m,
    ptrdiff_t *n,
    double *a,
    ptrdiff_t *lda,
    double *tau,
    double *work,
    ptrdiff_t *info
);

/* Source: zgeqr2p.f */
#define zgeqr2p FORTRAN_WRAPPER(zgeqr2p)
extern void zgeqr2p(
    ptrdiff_t *m,
    ptrdiff_t *n,
    double *a,
    ptrdiff_t *lda,
    double *tau,
    double *work,
    ptrdiff_t *info
);

/* Source: zgeqrf.f */
#define zgeqrf FORTRAN_WRAPPER(zgeqrf)
extern void zgeqrf(
    ptrdiff_t *m,
    ptrdiff_t *n,
    double *a,
    ptrdiff_t *lda,
    double *tau,
    double *work,
    ptrdiff_t *lwork,
    ptrdiff_t *info
);

/* Source: zgeqrfp.f */
#define zgeqrfp FORTRAN_WRAPPER(zgeqrfp)
extern void zgeqrfp(
    ptrdiff_t *m,
    ptrdiff_t *n,
    double *a,
    ptrdiff_t *lda,
    double *tau,
    double *work,
    ptrdiff_t *lwork,
    ptrdiff_t *info
);

/* Source: zgerfs.f */
#define zgerfs FORTRAN_WRAPPER(zgerfs)
extern void zgerfs(
    char   *trans,
    ptrdiff_t *n,
    ptrdiff_t *nrhs,
    double *a,
    ptrdiff_t *lda,
    double *af,
    ptrdiff_t *ldaf,
    ptrdiff_t *ipiv,
    double *b,
    ptrdiff_t *ldb,
    double *x,
    ptrdiff_t *ldx,
    double *ferr,
    double *berr,
    double *work,
    double *rwork,
    ptrdiff_t *info
);

/* Source: zgerq2.f */
#define zgerq2 FORTRAN_WRAPPER(zgerq2)
extern void zgerq2(
    ptrdiff_t *m,
    ptrdiff_t *n,
    double *a,
    ptrdiff_t *lda,
    double *tau,
    double *work,
    ptrdiff_t *info
);

/* Source: zgerqf.f */
#define zgerqf FORTRAN_WRAPPER(zgerqf)
extern void zgerqf(
    ptrdiff_t *m,
    ptrdiff_t *n,
    double *a,
    ptrdiff_t *lda,
    double *tau,
    double *work,
    ptrdiff_t *lwork,
    ptrdiff_t *info
);

/* Source: zgesc2.f */
#define zgesc2 FORTRAN_WRAPPER(zgesc2)
extern void zgesc2(
    ptrdiff_t *n,
    double *a,
    ptrdiff_t *lda,
    double *rhs,
    ptrdiff_t *ipiv,
    ptrdiff_t *jpiv,
    double *scale
);

/* Source: zgesdd.f */
#define zgesdd FORTRAN_WRAPPER(zgesdd)
extern void zgesdd(
    char   *jobz,
    ptrdiff_t *m,
    ptrdiff_t *n,
    double *a,
    ptrdiff_t *lda,
    double *s,
    double *u,
    ptrdiff_t *ldu,
    double *vt,
    ptrdiff_t *ldvt,
    double *work,
    ptrdiff_t *lwork,
    double *rwork,
    ptrdiff_t *iwork,
    ptrdiff_t *info
);

/* Source: zgesv.f */
#define zgesv FORTRAN_WRAPPER(zgesv)
extern void zgesv(
    ptrdiff_t *n,
    ptrdiff_t *nrhs,
    double *a,
    ptrdiff_t *lda,
    ptrdiff_t *ipiv,
    double *b,
    ptrdiff_t *ldb,
    ptrdiff_t *info
);

/* Source: zgesvd.f */
#define zgesvd FORTRAN_WRAPPER(zgesvd)
extern void zgesvd(
    char   *jobu,
    char   *jobvt,
    ptrdiff_t *m,
    ptrdiff_t *n,
    double *a,
    ptrdiff_t *lda,
    double *s,
    double *u,
    ptrdiff_t *ldu,
    double *vt,
    ptrdiff_t *ldvt,
    double *work,
    ptrdiff_t *lwork,
    double *rwork,
    ptrdiff_t *info
);

/* Source: zgesvx.f */
#define zgesvx FORTRAN_WRAPPER(zgesvx)
extern void zgesvx(
    char   *fact,
    char   *trans,
    ptrdiff_t *n,
    ptrdiff_t *nrhs,
    double *a,
    ptrdiff_t *lda,
    double *af,
    ptrdiff_t *ldaf,
    ptrdiff_t *ipiv,
    char   *equed,
    double *r,
    double *c,
    double *b,
    ptrdiff_t *ldb,
    double *x,
    ptrdiff_t *ldx,
    double *rcond,
    double *ferr,
    double *berr,
    double *work,
    double *rwork,
    ptrdiff_t *info
);

/* Source: zgetc2.f */
#define zgetc2 FORTRAN_WRAPPER(zgetc2)
extern void zgetc2(
    ptrdiff_t *n,
    double *a,
    ptrdiff_t *lda,
    ptrdiff_t *ipiv,
    ptrdiff_t *jpiv,
    ptrdiff_t *info
);

/* Source: zgetf2.f */
#define zgetf2 FORTRAN_WRAPPER(zgetf2)
extern void zgetf2(
    ptrdiff_t *m,
    ptrdiff_t *n,
    double *a,
    ptrdiff_t *lda,
    ptrdiff_t *ipiv,
    ptrdiff_t *info
);

/* Source: zgetrf.f */
#define zgetrf FORTRAN_WRAPPER(zgetrf)
extern void zgetrf(
    ptrdiff_t *m,
    ptrdiff_t *n,
    double *a,
    ptrdiff_t *lda,
    ptrdiff_t *ipiv,
    ptrdiff_t *info
);

/* Source: zgetri.f */
#define zgetri FORTRAN_WRAPPER(zgetri)
extern void zgetri(
    ptrdiff_t *n,
    double *a,
    ptrdiff_t *lda,
    ptrdiff_t *ipiv,
    double *work,
    ptrdiff_t *lwork,
    ptrdiff_t *info
);

/* Source: zgetrs.f */
#define zgetrs FORTRAN_WRAPPER(zgetrs)
extern void zgetrs(
    char   *trans,
    ptrdiff_t *n,
    ptrdiff_t *nrhs,
    double *a,
    ptrdiff_t *lda,
    ptrdiff_t *ipiv,
    double *b,
    ptrdiff_t *ldb,
    ptrdiff_t *info
);

/* Source: zggbak.f */
#define zggbak FORTRAN_WRAPPER(zggbak)
extern void zggbak(
    char   *job,
    char   *side,
    ptrdiff_t *n,
    ptrdiff_t *ilo,
    ptrdiff_t *ihi,
    double *lscale,
    double *rscale,
    ptrdiff_t *m,
    double *v,
    ptrdiff_t *ldv,
    ptrdiff_t *info
);

/* Source: zggbal.f */
#define zggbal FORTRAN_WRAPPER(zggbal)
extern void zggbal(
    char   *job,
    ptrdiff_t *n,
    double *a,
    ptrdiff_t *lda,
    double *b,
    ptrdiff_t *ldb,
    ptrdiff_t *ilo,
    ptrdiff_t *ihi,
    double *lscale,
    double *rscale,
    double *work,
    ptrdiff_t *info
);

/* Source: zgges.f */
#define zgges FORTRAN_WRAPPER(zgges)
extern void zgges(
    char   *jobvsl,
    char   *jobvsr,
    char   *sort,
    ptrdiff_t (*selctg)(),
    ptrdiff_t *n,
    double *a,
    ptrdiff_t *lda,
    double *b,
    ptrdiff_t *ldb,
    ptrdiff_t *sdim,
    double *alpha,
    double *beta,
    double *vsl,
    ptrdiff_t *ldvsl,
    double *vsr,
    ptrdiff_t *ldvsr,
    double *work,
    ptrdiff_t *lwork,
    double *rwork,
    ptrdiff_t *bwork,
    ptrdiff_t *info
);

/* Source: zggesx.f */
#define zggesx FORTRAN_WRAPPER(zggesx)
extern void zggesx(
    char   *jobvsl,
    char   *jobvsr,
    char   *sort,
    ptrdiff_t (*selctg)(),
    char   *sense,
    ptrdiff_t *n,
    double *a,
    ptrdiff_t *lda,
    double *b,
    ptrdiff_t *ldb,
    ptrdiff_t *sdim,
    double *alpha,
    double *beta,
    double *vsl,
    ptrdiff_t *ldvsl,
    double *vsr,
    ptrdiff_t *ldvsr,
    double *rconde,
    double *rcondv,
    double *work,
    ptrdiff_t *lwork,
    double *rwork,
    ptrdiff_t *iwork,
    ptrdiff_t *liwork,
    ptrdiff_t *bwork,
    ptrdiff_t *info
);

/* Source: zggev.f */
#define zggev FORTRAN_WRAPPER(zggev)
extern void zggev(
    char   *jobvl,
    char   *jobvr,
    ptrdiff_t *n,
    double *a,
    ptrdiff_t *lda,
    double *b,
    ptrdiff_t *ldb,
    double *alpha,
    double *beta,
    double *vl,
    ptrdiff_t *ldvl,
    double *vr,
    ptrdiff_t *ldvr,
    double *work,
    ptrdiff_t *lwork,
    double *rwork,
    ptrdiff_t *info
);

/* Source: zggevx.f */
#define zggevx FORTRAN_WRAPPER(zggevx)
extern void zggevx(
    char   *balanc,
    char   *jobvl,
    char   *jobvr,
    char   *sense,
    ptrdiff_t *n,
    double *a,
    ptrdiff_t *lda,
    double *b,
    ptrdiff_t *ldb,
    double *alpha,
    double *beta,
    double *vl,
    ptrdiff_t *ldvl,
    double *vr,
    ptrdiff_t *ldvr,
    ptrdiff_t *ilo,
    ptrdiff_t *ihi,
    double *lscale,
    double *rscale,
    double *abnrm,
    double *bbnrm,
    double *rconde,
    double *rcondv,
    double *work,
    ptrdiff_t *lwork,
    double *rwork,
    ptrdiff_t *iwork,
    ptrdiff_t *bwork,
    ptrdiff_t *info
);

/* Source: zggglm.f */
#define zggglm FORTRAN_WRAPPER(zggglm)
extern void zggglm(
    ptrdiff_t *n,
    ptrdiff_t *m,
    ptrdiff_t *p,
    double *a,
    ptrdiff_t *lda,
    double *b,
    ptrdiff_t *ldb,
    double *d,
    double *x,
    double *y,
    double *work,
    ptrdiff_t *lwork,
    ptrdiff_t *info
);

/* Source: zgghrd.f */
#define zgghrd FORTRAN_WRAPPER(zgghrd)
extern void zgghrd(
    char   *compq,
    char   *compz,
    ptrdiff_t *n,
    ptrdiff_t *ilo,
    ptrdiff_t *ihi,
    double *a,
    ptrdiff_t *lda,
    double *b,
    ptrdiff_t *ldb,
    double *q,
    ptrdiff_t *ldq,
    double *z,
    ptrdiff_t *ldz,
    ptrdiff_t *info
);

/* Source: zgglse.f */
#define zgglse FORTRAN_WRAPPER(zgglse)
extern void zgglse(
    ptrdiff_t *m,
    ptrdiff_t *n,
    ptrdiff_t *p,
    double *a,
    ptrdiff_t *lda,
    double *b,
    ptrdiff_t *ldb,
    double *c,
    double *d,
    double *x,
    double *work,
    ptrdiff_t *lwork,
    ptrdiff_t *info
);

/* Source: zggqrf.f */
#define zggqrf FORTRAN_WRAPPER(zggqrf)
extern void zggqrf(
    ptrdiff_t *n,
    ptrdiff_t *m,
    ptrdiff_t *p,
    double *a,
    ptrdiff_t *lda,
    double *taua,
    double *b,
    ptrdiff_t *ldb,
    double *taub,
    double *work,
    ptrdiff_t *lwork,
    ptrdiff_t *info
);

/* Source: zggrqf.f */
#define zggrqf FORTRAN_WRAPPER(zggrqf)
extern void zggrqf(
    ptrdiff_t *m,
    ptrdiff_t *p,
    ptrdiff_t *n,
    double *a,
    ptrdiff_t *lda,
    double *taua,
    double *b,
    ptrdiff_t *ldb,
    double *taub,
    double *work,
    ptrdiff_t *lwork,
    ptrdiff_t *info
);

/* Source: zggsvd.f */
#define zggsvd FORTRAN_WRAPPER(zggsvd)
extern void zggsvd(
    char   *jobu,
    char   *jobv,
    char   *jobq,
    ptrdiff_t *m,
    ptrdiff_t *n,
    ptrdiff_t *p,
    ptrdiff_t *k,
    ptrdiff_t *l,
    double *a,
    ptrdiff_t *lda,
    double *b,
    ptrdiff_t *ldb,
    double *alpha,
    double *beta,
    double *u,
    ptrdiff_t *ldu,
    double *v,
    ptrdiff_t *ldv,
    double *q,
    ptrdiff_t *ldq,
    double *work,
    double *rwork,
    ptrdiff_t *iwork,
    ptrdiff_t *info
);

/* Source: zggsvp.f */
#define zggsvp FORTRAN_WRAPPER(zggsvp)
extern void zggsvp(
    char   *jobu,
    char   *jobv,
    char   *jobq,
    ptrdiff_t *m,
    ptrdiff_t *p,
    ptrdiff_t *n,
    double *a,
    ptrdiff_t *lda,
    double *b,
    ptrdiff_t *ldb,
    double *tola,
    double *tolb,
    ptrdiff_t *k,
    ptrdiff_t *l,
    double *u,
    ptrdiff_t *ldu,
    double *v,
    ptrdiff_t *ldv,
    double *q,
    ptrdiff_t *ldq,
    ptrdiff_t *iwork,
    double *rwork,
    double *tau,
    double *work,
    ptrdiff_t *info
);

/* Source: zgtcon.f */
#define zgtcon FORTRAN_WRAPPER(zgtcon)
extern void zgtcon(
    char   *norm,
    ptrdiff_t *n,
    double *dl,
    double *d,
    double *du,
    double *du2,
    ptrdiff_t *ipiv,
    double *anorm,
    double *rcond,
    double *work,
    ptrdiff_t *info
);

/* Source: zgtrfs.f */
#define zgtrfs FORTRAN_WRAPPER(zgtrfs)
extern void zgtrfs(
    char   *trans,
    ptrdiff_t *n,
    ptrdiff_t *nrhs,
    double *dl,
    double *d,
    double *du,
    double *dlf,
    double *df,
    double *duf,
    double *du2,
    ptrdiff_t *ipiv,
    double *b,
    ptrdiff_t *ldb,
    double *x,
    ptrdiff_t *ldx,
    double *ferr,
    double *berr,
    double *work,
    double *rwork,
    ptrdiff_t *info
);

/* Source: zgtsv.f */
#define zgtsv FORTRAN_WRAPPER(zgtsv)
extern void zgtsv(
    ptrdiff_t *n,
    ptrdiff_t *nrhs,
    double *dl,
    double *d,
    double *du,
    double *b,
    ptrdiff_t *ldb,
    ptrdiff_t *info
);

/* Source: zgtsvx.f */
#define zgtsvx FORTRAN_WRAPPER(zgtsvx)
extern void zgtsvx(
    char   *fact,
    char   *trans,
    ptrdiff_t *n,
    ptrdiff_t *nrhs,
    double *dl,
    double *d,
    double *du,
    double *dlf,
    double *df,
    double *duf,
    double *du2,
    ptrdiff_t *ipiv,
    double *b,
    ptrdiff_t *ldb,
    double *x,
    ptrdiff_t *ldx,
    double *rcond,
    double *ferr,
    double *berr,
    double *work,
    double *rwork,
    ptrdiff_t *info
);

/* Source: zgttrf.f */
#define zgttrf FORTRAN_WRAPPER(zgttrf)
extern void zgttrf(
    ptrdiff_t *n,
    double *dl,
    double *d,
    double *du,
    double *du2,
    ptrdiff_t *ipiv,
    ptrdiff_t *info
);

/* Source: zgttrs.f */
#define zgttrs FORTRAN_WRAPPER(zgttrs)
extern void zgttrs(
    char   *trans,
    ptrdiff_t *n,
    ptrdiff_t *nrhs,
    double *dl,
    double *d,
    double *du,
    double *du2,
    ptrdiff_t *ipiv,
    double *b,
    ptrdiff_t *ldb,
    ptrdiff_t *info
);

/* Source: zgtts2.f */
#define zgtts2 FORTRAN_WRAPPER(zgtts2)
extern void zgtts2(
    ptrdiff_t *itrans,
    ptrdiff_t *n,
    ptrdiff_t *nrhs,
    double *dl,
    double *d,
    double *du,
    double *du2,
    ptrdiff_t *ipiv,
    double *b,
    ptrdiff_t *ldb
);

/* Source: zhbev.f */
#define zhbev FORTRAN_WRAPPER(zhbev)
extern void zhbev(
    char   *jobz,
    char   *uplo,
    ptrdiff_t *n,
    ptrdiff_t *kd,
    double *ab,
    ptrdiff_t *ldab,
    double *w,
    double *z,
    ptrdiff_t *ldz,
    double *work,
    double *rwork,
    ptrdiff_t *info
);

/* Source: zhbevd.f */
#define zhbevd FORTRAN_WRAPPER(zhbevd)
extern void zhbevd(
    char   *jobz,
    char   *uplo,
    ptrdiff_t *n,
    ptrdiff_t *kd,
    double *ab,
    ptrdiff_t *ldab,
    double *w,
    double *z,
    ptrdiff_t *ldz,
    double *work,
    ptrdiff_t *lwork,
    double *rwork,
    ptrdiff_t *lrwork,
    ptrdiff_t *iwork,
    ptrdiff_t *liwork,
    ptrdiff_t *info
);

/* Source: zhbevx.f */
#define zhbevx FORTRAN_WRAPPER(zhbevx)
extern void zhbevx(
    char   *jobz,
    char   *range,
    char   *uplo,
    ptrdiff_t *n,
    ptrdiff_t *kd,
    double *ab,
    ptrdiff_t *ldab,
    double *q,
    ptrdiff_t *ldq,
    double *vl,
    double *vu,
    ptrdiff_t *il,
    ptrdiff_t *iu,
    double *abstol,
    ptrdiff_t *m,
    double *w,
    double *z,
    ptrdiff_t *ldz,
    double *work,
    double *rwork,
    ptrdiff_t *iwork,
    ptrdiff_t *ifail,
    ptrdiff_t *info
);

/* Source: zhbgst.f */
#define zhbgst FORTRAN_WRAPPER(zhbgst)
extern void zhbgst(
    char   *vect,
    char   *uplo,
    ptrdiff_t *n,
    ptrdiff_t *ka,
    ptrdiff_t *kb,
    double *ab,
    ptrdiff_t *ldab,
    double *bb,
    ptrdiff_t *ldbb,
    double *x,
    ptrdiff_t *ldx,
    double *work,
    double *rwork,
    ptrdiff_t *info
);

/* Source: zhbgv.f */
#define zhbgv FORTRAN_WRAPPER(zhbgv)
extern void zhbgv(
    char   *jobz,
    char   *uplo,
    ptrdiff_t *n,
    ptrdiff_t *ka,
    ptrdiff_t *kb,
    double *ab,
    ptrdiff_t *ldab,
    double *bb,
    ptrdiff_t *ldbb,
    double *w,
    double *z,
    ptrdiff_t *ldz,
    double *work,
    double *rwork,
    ptrdiff_t *info
);

/* Source: zhbgvd.f */
#define zhbgvd FORTRAN_WRAPPER(zhbgvd)
extern void zhbgvd(
    char   *jobz,
    char   *uplo,
    ptrdiff_t *n,
    ptrdiff_t *ka,
    ptrdiff_t *kb,
    double *ab,
    ptrdiff_t *ldab,
    double *bb,
    ptrdiff_t *ldbb,
    double *w,
    double *z,
    ptrdiff_t *ldz,
    double *work,
    ptrdiff_t *lwork,
    double *rwork,
    ptrdiff_t *lrwork,
    ptrdiff_t *iwork,
    ptrdiff_t *liwork,
    ptrdiff_t *info
);

/* Source: zhbgvx.f */
#define zhbgvx FORTRAN_WRAPPER(zhbgvx)
extern void zhbgvx(
    char   *jobz,
    char   *range,
    char   *uplo,
    ptrdiff_t *n,
    ptrdiff_t *ka,
    ptrdiff_t *kb,
    double *ab,
    ptrdiff_t *ldab,
    double *bb,
    ptrdiff_t *ldbb,
    double *q,
    ptrdiff_t *ldq,
    double *vl,
    double *vu,
    ptrdiff_t *il,
    ptrdiff_t *iu,
    double *abstol,
    ptrdiff_t *m,
    double *w,
    double *z,
    ptrdiff_t *ldz,
    double *work,
    double *rwork,
    ptrdiff_t *iwork,
    ptrdiff_t *ifail,
    ptrdiff_t *info
);

/* Source: zhbtrd.f */
#define zhbtrd FORTRAN_WRAPPER(zhbtrd)
extern void zhbtrd(
    char   *vect,
    char   *uplo,
    ptrdiff_t *n,
    ptrdiff_t *kd,
    double *ab,
    ptrdiff_t *ldab,
    double *d,
    double *e,
    double *q,
    ptrdiff_t *ldq,
    double *work,
    ptrdiff_t *info
);

/* Source: zhecon.f */
#define zhecon FORTRAN_WRAPPER(zhecon)
extern void zhecon(
    char   *uplo,
    ptrdiff_t *n,
    double *a,
    ptrdiff_t *lda,
    ptrdiff_t *ipiv,
    double *anorm,
    double *rcond,
    double *work,
    ptrdiff_t *info
);

/* Source: zheequb.f */
#define zheequb FORTRAN_WRAPPER(zheequb)
extern void zheequb(
    char   *uplo,
    ptrdiff_t *n,
    double *a,
    ptrdiff_t *lda,
    double *s,
    double *scond,
    double *amax,
    double *work,
    ptrdiff_t *info
);

/* Source: zheev.f */
#define zheev FORTRAN_WRAPPER(zheev)
extern void zheev(
    char   *jobz,
    char   *uplo,
    ptrdiff_t *n,
    double *a,
    ptrdiff_t *lda,
    double *w,
    double *work,
    ptrdiff_t *lwork,
    double *rwork,
    ptrdiff_t *info
);

/* Source: zheevd.f */
#define zheevd FORTRAN_WRAPPER(zheevd)
extern void zheevd(
    char   *jobz,
    char   *uplo,
    ptrdiff_t *n,
    double *a,
    ptrdiff_t *lda,
    double *w,
    double *work,
    ptrdiff_t *lwork,
    double *rwork,
    ptrdiff_t *lrwork,
    ptrdiff_t *iwork,
    ptrdiff_t *liwork,
    ptrdiff_t *info
);

/* Source: zheevr.f */
#define zheevr FORTRAN_WRAPPER(zheevr)
extern void zheevr(
    char   *jobz,
    char   *range,
    char   *uplo,
    ptrdiff_t *n,
    double *a,
    ptrdiff_t *lda,
    double *vl,
    double *vu,
    ptrdiff_t *il,
    ptrdiff_t *iu,
    double *abstol,
    ptrdiff_t *m,
    double *w,
    double *z,
    ptrdiff_t *ldz,
    ptrdiff_t *isuppz,
    double *work,
    ptrdiff_t *lwork,
    double *rwork,
    ptrdiff_t *lrwork,
    ptrdiff_t *iwork,
    ptrdiff_t *liwork,
    ptrdiff_t *info
);

/* Source: zheevx.f */
#define zheevx FORTRAN_WRAPPER(zheevx)
extern void zheevx(
    char   *jobz,
    char   *range,
    char   *uplo,
    ptrdiff_t *n,
    double *a,
    ptrdiff_t *lda,
    double *vl,
    double *vu,
    ptrdiff_t *il,
    ptrdiff_t *iu,
    double *abstol,
    ptrdiff_t *m,
    double *w,
    double *z,
    ptrdiff_t *ldz,
    double *work,
    ptrdiff_t *lwork,
    double *rwork,
    ptrdiff_t *iwork,
    ptrdiff_t *ifail,
    ptrdiff_t *info
);

/* Source: zhegs2.f */
#define zhegs2 FORTRAN_WRAPPER(zhegs2)
extern void zhegs2(
    ptrdiff_t *itype,
    char   *uplo,
    ptrdiff_t *n,
    double *a,
    ptrdiff_t *lda,
    double *b,
    ptrdiff_t *ldb,
    ptrdiff_t *info
);

/* Source: zhegst.f */
#define zhegst FORTRAN_WRAPPER(zhegst)
extern void zhegst(
    ptrdiff_t *itype,
    char   *uplo,
    ptrdiff_t *n,
    double *a,
    ptrdiff_t *lda,
    double *b,
    ptrdiff_t *ldb,
    ptrdiff_t *info
);

/* Source: zhegv.f */
#define zhegv FORTRAN_WRAPPER(zhegv)
extern void zhegv(
    ptrdiff_t *itype,
    char   *jobz,
    char   *uplo,
    ptrdiff_t *n,
    double *a,
    ptrdiff_t *lda,
    double *b,
    ptrdiff_t *ldb,
    double *w,
    double *work,
    ptrdiff_t *lwork,
    double *rwork,
    ptrdiff_t *info
);

/* Source: zhegvd.f */
#define zhegvd FORTRAN_WRAPPER(zhegvd)
extern void zhegvd(
    ptrdiff_t *itype,
    char   *jobz,
    char   *uplo,
    ptrdiff_t *n,
    double *a,
    ptrdiff_t *lda,
    double *b,
    ptrdiff_t *ldb,
    double *w,
    double *work,
    ptrdiff_t *lwork,
    double *rwork,
    ptrdiff_t *lrwork,
    ptrdiff_t *iwork,
    ptrdiff_t *liwork,
    ptrdiff_t *info
);

/* Source: zhegvx.f */
#define zhegvx FORTRAN_WRAPPER(zhegvx)
extern void zhegvx(
    ptrdiff_t *itype,
    char   *jobz,
    char   *range,
    char   *uplo,
    ptrdiff_t *n,
    double *a,
    ptrdiff_t *lda,
    double *b,
    ptrdiff_t *ldb,
    double *vl,
    double *vu,
    ptrdiff_t *il,
    ptrdiff_t *iu,
    double *abstol,
    ptrdiff_t *m,
    double *w,
    double *z,
    ptrdiff_t *ldz,
    double *work,
    ptrdiff_t *lwork,
    double *rwork,
    ptrdiff_t *iwork,
    ptrdiff_t *ifail,
    ptrdiff_t *info
);

/* Source: zherfs.f */
#define zherfs FORTRAN_WRAPPER(zherfs)
extern void zherfs(
    char   *uplo,
    ptrdiff_t *n,
    ptrdiff_t *nrhs,
    double *a,
    ptrdiff_t *lda,
    double *af,
    ptrdiff_t *ldaf,
    ptrdiff_t *ipiv,
    double *b,
    ptrdiff_t *ldb,
    double *x,
    ptrdiff_t *ldx,
    double *ferr,
    double *berr,
    double *work,
    double *rwork,
    ptrdiff_t *info
);

/* Source: zhesv.f */
#define zhesv FORTRAN_WRAPPER(zhesv)
extern void zhesv(
    char   *uplo,
    ptrdiff_t *n,
    ptrdiff_t *nrhs,
    double *a,
    ptrdiff_t *lda,
    ptrdiff_t *ipiv,
    double *b,
    ptrdiff_t *ldb,
    double *work,
    ptrdiff_t *lwork,
    ptrdiff_t *info
);

/* Source: zhesvx.f */
#define zhesvx FORTRAN_WRAPPER(zhesvx)
extern void zhesvx(
    char   *fact,
    char   *uplo,
    ptrdiff_t *n,
    ptrdiff_t *nrhs,
    double *a,
    ptrdiff_t *lda,
    double *af,
    ptrdiff_t *ldaf,
    ptrdiff_t *ipiv,
    double *b,
    ptrdiff_t *ldb,
    double *x,
    ptrdiff_t *ldx,
    double *rcond,
    double *ferr,
    double *berr,
    double *work,
    ptrdiff_t *lwork,
    double *rwork,
    ptrdiff_t *info
);

/* Source: zhetd2.f */
#define zhetd2 FORTRAN_WRAPPER(zhetd2)
extern void zhetd2(
    char   *uplo,
    ptrdiff_t *n,
    double *a,
    ptrdiff_t *lda,
    double *d,
    double *e,
    double *tau,
    ptrdiff_t *info
);

/* Source: zhetf2.f */
#define zhetf2 FORTRAN_WRAPPER(zhetf2)
extern void zhetf2(
    char   *uplo,
    ptrdiff_t *n,
    double *a,
    ptrdiff_t *lda,
    ptrdiff_t *ipiv,
    ptrdiff_t *info
);

/* Source: zhetrd.f */
#define zhetrd FORTRAN_WRAPPER(zhetrd)
extern void zhetrd(
    char   *uplo,
    ptrdiff_t *n,
    double *a,
    ptrdiff_t *lda,
    double *d,
    double *e,
    double *tau,
    double *work,
    ptrdiff_t *lwork,
    ptrdiff_t *info
);

/* Source: zhetrf.f */
#define zhetrf FORTRAN_WRAPPER(zhetrf)
extern void zhetrf(
    char   *uplo,
    ptrdiff_t *n,
    double *a,
    ptrdiff_t *lda,
    ptrdiff_t *ipiv,
    double *work,
    ptrdiff_t *lwork,
    ptrdiff_t *info
);

/* Source: zhetri.f */
#define zhetri FORTRAN_WRAPPER(zhetri)
extern void zhetri(
    char   *uplo,
    ptrdiff_t *n,
    double *a,
    ptrdiff_t *lda,
    ptrdiff_t *ipiv,
    double *work,
    ptrdiff_t *info
);

/* Source: zhetrs.f */
#define zhetrs FORTRAN_WRAPPER(zhetrs)
extern void zhetrs(
    char   *uplo,
    ptrdiff_t *n,
    ptrdiff_t *nrhs,
    double *a,
    ptrdiff_t *lda,
    ptrdiff_t *ipiv,
    double *b,
    ptrdiff_t *ldb,
    ptrdiff_t *info
);

/* Source: zhfrk.f */
#define zhfrk FORTRAN_WRAPPER(zhfrk)
extern void zhfrk(
    char   *transr,
    char   *uplo,
    char   *trans,
    ptrdiff_t *n,
    ptrdiff_t *k,
    double *alpha,
    double *a,
    ptrdiff_t *lda,
    double *beta,
    double *c
);

/* Source: zhgeqz.f */
#define zhgeqz FORTRAN_WRAPPER(zhgeqz)
extern void zhgeqz(
    char   *job,
    char   *compq,
    char   *compz,
    ptrdiff_t *n,
    ptrdiff_t *ilo,
    ptrdiff_t *ihi,
    double *h,
    ptrdiff_t *ldh,
    double *t,
    ptrdiff_t *ldt,
    double *alpha,
    double *beta,
    double *q,
    ptrdiff_t *ldq,
    double *z,
    ptrdiff_t *ldz,
    double *work,
    ptrdiff_t *lwork,
    double *rwork,
    ptrdiff_t *info
);

/* Source: zhpcon.f */
#define zhpcon FORTRAN_WRAPPER(zhpcon)
extern void zhpcon(
    char   *uplo,
    ptrdiff_t *n,
    double *ap,
    ptrdiff_t *ipiv,
    double *anorm,
    double *rcond,
    double *work,
    ptrdiff_t *info
);

/* Source: zhpev.f */
#define zhpev FORTRAN_WRAPPER(zhpev)
extern void zhpev(
    char   *jobz,
    char   *uplo,
    ptrdiff_t *n,
    double *ap,
    double *w,
    double *z,
    ptrdiff_t *ldz,
    double *work,
    double *rwork,
    ptrdiff_t *info
);

/* Source: zhpevd.f */
#define zhpevd FORTRAN_WRAPPER(zhpevd)
extern void zhpevd(
    char   *jobz,
    char   *uplo,
    ptrdiff_t *n,
    double *ap,
    double *w,
    double *z,
    ptrdiff_t *ldz,
    double *work,
    ptrdiff_t *lwork,
    double *rwork,
    ptrdiff_t *lrwork,
    ptrdiff_t *iwork,
    ptrdiff_t *liwork,
    ptrdiff_t *info
);

/* Source: zhpevx.f */
#define zhpevx FORTRAN_WRAPPER(zhpevx)
extern void zhpevx(
    char   *jobz,
    char   *range,
    char   *uplo,
    ptrdiff_t *n,
    double *ap,
    double *vl,
    double *vu,
    ptrdiff_t *il,
    ptrdiff_t *iu,
    double *abstol,
    ptrdiff_t *m,
    double *w,
    double *z,
    ptrdiff_t *ldz,
    double *work,
    double *rwork,
    ptrdiff_t *iwork,
    ptrdiff_t *ifail,
    ptrdiff_t *info
);

/* Source: zhpgst.f */
#define zhpgst FORTRAN_WRAPPER(zhpgst)
extern void zhpgst(
    ptrdiff_t *itype,
    char   *uplo,
    ptrdiff_t *n,
    double *ap,
    double *bp,
    ptrdiff_t *info
);

/* Source: zhpgv.f */
#define zhpgv FORTRAN_WRAPPER(zhpgv)
extern void zhpgv(
    ptrdiff_t *itype,
    char   *jobz,
    char   *uplo,
    ptrdiff_t *n,
    double *ap,
    double *bp,
    double *w,
    double *z,
    ptrdiff_t *ldz,
    double *work,
    double *rwork,
    ptrdiff_t *info
);

/* Source: zhpgvd.f */
#define zhpgvd FORTRAN_WRAPPER(zhpgvd)
extern void zhpgvd(
    ptrdiff_t *itype,
    char   *jobz,
    char   *uplo,
    ptrdiff_t *n,
    double *ap,
    double *bp,
    double *w,
    double *z,
    ptrdiff_t *ldz,
    double *work,
    ptrdiff_t *lwork,
    double *rwork,
    ptrdiff_t *lrwork,
    ptrdiff_t *iwork,
    ptrdiff_t *liwork,
    ptrdiff_t *info
);

/* Source: zhpgvx.f */
#define zhpgvx FORTRAN_WRAPPER(zhpgvx)
extern void zhpgvx(
    ptrdiff_t *itype,
    char   *jobz,
    char   *range,
    char   *uplo,
    ptrdiff_t *n,
    double *ap,
    double *bp,
    double *vl,
    double *vu,
    ptrdiff_t *il,
    ptrdiff_t *iu,
    double *abstol,
    ptrdiff_t *m,
    double *w,
    double *z,
    ptrdiff_t *ldz,
    double *work,
    double *rwork,
    ptrdiff_t *iwork,
    ptrdiff_t *ifail,
    ptrdiff_t *info
);

/* Source: zhprfs.f */
#define zhprfs FORTRAN_WRAPPER(zhprfs)
extern void zhprfs(
    char   *uplo,
    ptrdiff_t *n,
    ptrdiff_t *nrhs,
    double *ap,
    double *afp,
    ptrdiff_t *ipiv,
    double *b,
    ptrdiff_t *ldb,
    double *x,
    ptrdiff_t *ldx,
    double *ferr,
    double *berr,
    double *work,
    double *rwork,
    ptrdiff_t *info
);

/* Source: zhpsv.f */
#define zhpsv FORTRAN_WRAPPER(zhpsv)
extern void zhpsv(
    char   *uplo,
    ptrdiff_t *n,
    ptrdiff_t *nrhs,
    double *ap,
    ptrdiff_t *ipiv,
    double *b,
    ptrdiff_t *ldb,
    ptrdiff_t *info
);

/* Source: zhpsvx.f */
#define zhpsvx FORTRAN_WRAPPER(zhpsvx)
extern void zhpsvx(
    char   *fact,
    char   *uplo,
    ptrdiff_t *n,
    ptrdiff_t *nrhs,
    double *ap,
    double *afp,
    ptrdiff_t *ipiv,
    double *b,
    ptrdiff_t *ldb,
    double *x,
    ptrdiff_t *ldx,
    double *rcond,
    double *ferr,
    double *berr,
    double *work,
    double *rwork,
    ptrdiff_t *info
);

/* Source: zhptrd.f */
#define zhptrd FORTRAN_WRAPPER(zhptrd)
extern void zhptrd(
    char   *uplo,
    ptrdiff_t *n,
    double *ap,
    double *d,
    double *e,
    double *tau,
    ptrdiff_t *info
);

/* Source: zhptrf.f */
#define zhptrf FORTRAN_WRAPPER(zhptrf)
extern void zhptrf(
    char   *uplo,
    ptrdiff_t *n,
    double *ap,
    ptrdiff_t *ipiv,
    ptrdiff_t *info
);

/* Source: zhptri.f */
#define zhptri FORTRAN_WRAPPER(zhptri)
extern void zhptri(
    char   *uplo,
    ptrdiff_t *n,
    double *ap,
    ptrdiff_t *ipiv,
    double *work,
    ptrdiff_t *info
);

/* Source: zhptrs.f */
#define zhptrs FORTRAN_WRAPPER(zhptrs)
extern void zhptrs(
    char   *uplo,
    ptrdiff_t *n,
    ptrdiff_t *nrhs,
    double *ap,
    ptrdiff_t *ipiv,
    double *b,
    ptrdiff_t *ldb,
    ptrdiff_t *info
);

/* Source: zhsein.f */
#define zhsein FORTRAN_WRAPPER(zhsein)
extern void zhsein(
    char   *side,
    char   *eigsrc,
    char   *initv,
    ptrdiff_t *select,
    ptrdiff_t *n,
    double *h,
    ptrdiff_t *ldh,
    double *w,
    double *vl,
    ptrdiff_t *ldvl,
    double *vr,
    ptrdiff_t *ldvr,
    ptrdiff_t *mm,
    ptrdiff_t *m,
    double *work,
    double *rwork,
    ptrdiff_t *ifaill,
    ptrdiff_t *ifailr,
    ptrdiff_t *info
);

/* Source: zhseqr.f */
#define zhseqr FORTRAN_WRAPPER(zhseqr)
extern void zhseqr(
    char   *job,
    char   *compz,
    ptrdiff_t *n,
    ptrdiff_t *ilo,
    ptrdiff_t *ihi,
    double *h,
    ptrdiff_t *ldh,
    double *w,
    double *z,
    ptrdiff_t *ldz,
    double *work,
    ptrdiff_t *lwork,
    ptrdiff_t *info
);

/* Source: zlabrd.f */
#define zlabrd FORTRAN_WRAPPER(zlabrd)
extern void zlabrd(
    ptrdiff_t *m,
    ptrdiff_t *n,
    ptrdiff_t *nb,
    double *a,
    ptrdiff_t *lda,
    double *d,
    double *e,
    double *tauq,
    double *taup,
    double *x,
    ptrdiff_t *ldx,
    double *y,
    ptrdiff_t *ldy
);

/* Source: zlacgv.f */
#define zlacgv FORTRAN_WRAPPER(zlacgv)
extern void zlacgv(
    ptrdiff_t *n,
    double *x,
    ptrdiff_t *incx
);

/* Source: zlacn2.f */
#define zlacn2 FORTRAN_WRAPPER(zlacn2)
extern void zlacn2(
    ptrdiff_t *n,
    double *v,
    double *x,
    double *est,
    ptrdiff_t *kase,
    ptrdiff_t *isave
);

/* Source: zlacon.f */
#define zlacon FORTRAN_WRAPPER(zlacon)
extern void zlacon(
    ptrdiff_t *n,
    double *v,
    double *x,
    double *est,
    ptrdiff_t *kase
);

/* Source: zlacp2.f */
#define zlacp2 FORTRAN_WRAPPER(zlacp2)
extern void zlacp2(
    char   *uplo,
    ptrdiff_t *m,
    ptrdiff_t *n,
    double *a,
    ptrdiff_t *lda,
    double *b,
    ptrdiff_t *ldb
);

/* Source: zlacpy.f */
#define zlacpy FORTRAN_WRAPPER(zlacpy)
extern void zlacpy(
    char   *uplo,
    ptrdiff_t *m,
    ptrdiff_t *n,
    double *a,
    ptrdiff_t *lda,
    double *b,
    ptrdiff_t *ldb
);

/* Source: zlacrm.f */
#define zlacrm FORTRAN_WRAPPER(zlacrm)
extern void zlacrm(
    ptrdiff_t *m,
    ptrdiff_t *n,
    double *a,
    ptrdiff_t *lda,
    double *b,
    ptrdiff_t *ldb,
    double *c,
    ptrdiff_t *ldc,
    double *rwork
);

/* Source: zlacrt.f */
#define zlacrt FORTRAN_WRAPPER(zlacrt)
extern void zlacrt(
    ptrdiff_t *n,
    double *cx,
    ptrdiff_t *incx,
    double *cy,
    ptrdiff_t *incy,
    double *c,
    double *s
);

/* Source: zladiv.f */
#define zladiv FORTRAN_WRAPPER(zladiv)
#ifndef FORTRAN_COMPLEX_FUNCTIONS_RETURN_VOID
extern doublecomplex zladiv(
#else
extern void zladiv(
    doublecomplex* retval,
#endif
    double *x,
    double *y
);

/* Source: zlaed0.f */
#define zlaed0 FORTRAN_WRAPPER(zlaed0)
extern void zlaed0(
    ptrdiff_t *qsiz,
    ptrdiff_t *n,
    double *d,
    double *e,
    double *q,
    ptrdiff_t *ldq,
    double *qstore,
    ptrdiff_t *ldqs,
    double *rwork,
    ptrdiff_t *iwork,
    ptrdiff_t *info
);

/* Source: zlaed7.f */
#define zlaed7 FORTRAN_WRAPPER(zlaed7)
extern void zlaed7(
    ptrdiff_t *n,
    ptrdiff_t *cutpnt,
    ptrdiff_t *qsiz,
    ptrdiff_t *tlvls,
    ptrdiff_t *curlvl,
    ptrdiff_t *curpbm,
    double *d,
    double *q,
    ptrdiff_t *ldq,
    double *rho,
    ptrdiff_t *indxq,
    double *qstore,
    ptrdiff_t *qptr,
    ptrdiff_t *prmptr,
    ptrdiff_t *perm,
    ptrdiff_t *givptr,
    ptrdiff_t *givcol,
    double *givnum,
    double *work,
    double *rwork,
    ptrdiff_t *iwork,
    ptrdiff_t *info
);

/* Source: zlaed8.f */
#define zlaed8 FORTRAN_WRAPPER(zlaed8)
extern void zlaed8(
    ptrdiff_t *k,
    ptrdiff_t *n,
    ptrdiff_t *qsiz,
    double *q,
    ptrdiff_t *ldq,
    double *d,
    double *rho,
    ptrdiff_t *cutpnt,
    double *z,
    double *dlamda,
    double *q2,
    ptrdiff_t *ldq2,
    double *w,
    ptrdiff_t *indxp,
    ptrdiff_t *indx,
    ptrdiff_t *indxq,
    ptrdiff_t *perm,
    ptrdiff_t *givptr,
    ptrdiff_t *givcol,
    double *givnum,
    ptrdiff_t *info
);

/* Source: zlaein.f */
#define zlaein FORTRAN_WRAPPER(zlaein)
extern void zlaein(
    ptrdiff_t *rightv,
    ptrdiff_t *noinit,
    ptrdiff_t *n,
    double *h,
    ptrdiff_t *ldh,
    double *w,
    double *v,
    double *b,
    ptrdiff_t *ldb,
    double *rwork,
    double *eps3,
    double *smlnum,
    ptrdiff_t *info
);

/* Source: zlaesy.f */
#define zlaesy FORTRAN_WRAPPER(zlaesy)
extern void zlaesy(
    double *a,
    double *b,
    double *c,
    double *rt1,
    double *rt2,
    double *evscal,
    double *cs1,
    double *sn1
);

/* Source: zlaev2.f */
#define zlaev2 FORTRAN_WRAPPER(zlaev2)
extern void zlaev2(
    double *a,
    double *b,
    double *c,
    double *rt1,
    double *rt2,
    double *cs1,
    double *sn1
);

/* Source: zlag2c.f */
#define zlag2c FORTRAN_WRAPPER(zlag2c)
extern void zlag2c(
    ptrdiff_t *m,
    ptrdiff_t *n,
    double *a,
    ptrdiff_t *lda,
    float  *sa,
    ptrdiff_t *ldsa,
    ptrdiff_t *info
);

/* Source: zlags2.f */
#define zlags2 FORTRAN_WRAPPER(zlags2)
extern void zlags2(
    ptrdiff_t *upper,
    double *a1,
    double *a2,
    double *a3,
    double *b1,
    double *b2,
    double *b3,
    double *csu,
    double *snu,
    double *csv,
    double *snv,
    double *csq,
    double *snq
);

/* Source: zlagtm.f */
#define zlagtm FORTRAN_WRAPPER(zlagtm)
extern void zlagtm(
    char   *trans,
    ptrdiff_t *n,
    ptrdiff_t *nrhs,
    double *alpha,
    double *dl,
    double *d,
    double *du,
    double *x,
    ptrdiff_t *ldx,
    double *beta,
    double *b,
    ptrdiff_t *ldb
);

/* Source: zlahef.f */
#define zlahef FORTRAN_WRAPPER(zlahef)
extern void zlahef(
    char   *uplo,
    ptrdiff_t *n,
    ptrdiff_t *nb,
    ptrdiff_t *kb,
    double *a,
    ptrdiff_t *lda,
    ptrdiff_t *ipiv,
    double *w,
    ptrdiff_t *ldw,
    ptrdiff_t *info
);

/* Source: zlahqr.f */
#define zlahqr FORTRAN_WRAPPER(zlahqr)
extern void zlahqr(
    ptrdiff_t *wantt,
    ptrdiff_t *wantz,
    ptrdiff_t *n,
    ptrdiff_t *ilo,
    ptrdiff_t *ihi,
    double *h,
    ptrdiff_t *ldh,
    double *w,
    ptrdiff_t *iloz,
    ptrdiff_t *ihiz,
    double *z,
    ptrdiff_t *ldz,
    ptrdiff_t *info
);

/* Source: zlahr2.f */
#define zlahr2 FORTRAN_WRAPPER(zlahr2)
extern void zlahr2(
    ptrdiff_t *n,
    ptrdiff_t *k,
    ptrdiff_t *nb,
    double *a,
    ptrdiff_t *lda,
    double *tau,
    double *t,
    ptrdiff_t *ldt,
    double *y,
    ptrdiff_t *ldy
);

/* Source: zlahrd.f */
#define zlahrd FORTRAN_WRAPPER(zlahrd)
extern void zlahrd(
    ptrdiff_t *n,
    ptrdiff_t *k,
    ptrdiff_t *nb,
    double *a,
    ptrdiff_t *lda,
    double *tau,
    double *t,
    ptrdiff_t *ldt,
    double *y,
    ptrdiff_t *ldy
);

/* Source: zlaic1.f */
#define zlaic1 FORTRAN_WRAPPER(zlaic1)
extern void zlaic1(
    ptrdiff_t *job,
    ptrdiff_t *j,
    double *x,
    double *sest,
    double *w,
    double *gamma_,
    double *sestpr,
    double *s,
    double *c
);

/* Source: zlals0.f */
#define zlals0 FORTRAN_WRAPPER(zlals0)
extern void zlals0(
    ptrdiff_t *icompq,
    ptrdiff_t *nl,
    ptrdiff_t *nr,
    ptrdiff_t *sqre,
    ptrdiff_t *nrhs,
    double *b,
    ptrdiff_t *ldb,
    double *bx,
    ptrdiff_t *ldbx,
    ptrdiff_t *perm,
    ptrdiff_t *givptr,
    ptrdiff_t *givcol,
    ptrdiff_t *ldgcol,
    double *givnum,
    ptrdiff_t *ldgnum,
    double *poles,
    double *difl,
    double *difr,
    double *z,
    ptrdiff_t *k,
    double *c,
    double *s,
    double *rwork,
    ptrdiff_t *info
);

/* Source: zlalsa.f */
#define zlalsa FORTRAN_WRAPPER(zlalsa)
extern void zlalsa(
    ptrdiff_t *icompq,
    ptrdiff_t *smlsiz,
    ptrdiff_t *n,
    ptrdiff_t *nrhs,
    double *b,
    ptrdiff_t *ldb,
    double *bx,
    ptrdiff_t *ldbx,
    double *u,
    ptrdiff_t *ldu,
    double *vt,
    ptrdiff_t *k,
    double *difl,
    double *difr,
    double *z,
    double *poles,
    ptrdiff_t *givptr,
    ptrdiff_t *givcol,
    ptrdiff_t *ldgcol,
    ptrdiff_t *perm,
    double *givnum,
    double *c,
    double *s,
    double *rwork,
    ptrdiff_t *iwork,
    ptrdiff_t *info
);

/* Source: zlalsd.f */
#define zlalsd FORTRAN_WRAPPER(zlalsd)
extern void zlalsd(
    char   *uplo,
    ptrdiff_t *smlsiz,
    ptrdiff_t *n,
    ptrdiff_t *nrhs,
    double *d,
    double *e,
    double *b,
    ptrdiff_t *ldb,
    double *rcond,
    ptrdiff_t *rank,
    double *work,
    double *rwork,
    ptrdiff_t *iwork,
    ptrdiff_t *info
);

/* Source: zlangb.f */
#define zlangb FORTRAN_WRAPPER(zlangb)
extern double zlangb(
    char   *norm,
    ptrdiff_t *n,
    ptrdiff_t *kl,
    ptrdiff_t *ku,
    double *ab,
    ptrdiff_t *ldab,
    double *work
);

/* Source: zlange.f */
#define zlange FORTRAN_WRAPPER(zlange)
extern double zlange(
    char   *norm,
    ptrdiff_t *m,
    ptrdiff_t *n,
    double *a,
    ptrdiff_t *lda,
    double *work
);

/* Source: zlangt.f */
#define zlangt FORTRAN_WRAPPER(zlangt)
extern double zlangt(
    char   *norm,
    ptrdiff_t *n,
    double *dl,
    double *d,
    double *du
);

/* Source: zlanhb.f */
#define zlanhb FORTRAN_WRAPPER(zlanhb)
extern double zlanhb(
    char   *norm,
    char   *uplo,
    ptrdiff_t *n,
    ptrdiff_t *k,
    double *ab,
    ptrdiff_t *ldab,
    double *work
);
```
